LIN {X 0,Y 427.231,Z 476.03,A -85,B 0,C 180,E1 9027.625,E2 9027.625} C_VEL
LIN {X 0,Y 427.048,Z 476.03,A -85,B 0,C 180,E1 9034.562,E2 9034.562} C_VEL
LIN {X 0,Y 427.063,Z 476.03,A -85,B 0,C 180,E1 9039.656,E2 9039.656} C_VEL
LIN {X 0,Y 427.079,Z 476.03,A -85,B 0,C 180,E1 9045.158,E2 9045.158} C_VEL
LIN {X 0,Y 427.044,Z 476.03,A -85,B 0,C 180,E1 9051.263,E2 9051.263} C_VEL
LIN {X 0,Y 427.131,Z 476.03,A -85,B 0,C 180,E1 9058.294,E2 9058.294} C_VEL
LIN {X 0,Y 427.346,Z 476.125,A -85,B 0,C 180,E1 9064.803,E2 9064.803} C_VEL
LIN {X 0,Y 433.891,Z 490.356,A -85,B 0,C 180,E1 9065.954,E2 9065.954} C_VEL
LIN {X 0,Y 447.35,Z 521.334,A -85,B 0,C 180,E1 9068.749,E2 9068.749} C_VEL
LIN {X 0,Y 452.812,Z 539.377,A -85,B 0,C 180,E1 9070.383,E2 9070.383} C_VEL
LIN {X 0,Y 448.1,Z 575.713,A -85,B 0,C 180,E1 9072.93,E2 9072.93} C_VEL
LIN {X 0,Y 442.863,Z 608.573,A -85,B 0,C 180,E1 9076.154,E2 9076.154} C_VEL
LIN {X 0,Y 438.068,Z 636.216,A -85,B 0,C 180,E1 9079.797,E2 9079.797} C_VEL
LIN {X 0,Y 434.006,Z 660.175,A -85,B 0,C 180,E1 9083.993,E2 9083.993} C_VEL
LIN {X 0,Y 431.161,Z 679.406,A -85,B 0,C 180,E1 9088.491,E2 9088.491} C_VEL
LIN {X 0,Y 429.325,Z 694.838,A -85,B 0,C 180,E1 9093.539,E2 9093.539} C_VEL
LIN {X 0,Y 428.567,Z 704.775,A -85,B 0,C 180,E1 9098.423,E2 9098.423} C_VEL
LIN {X 0,Y 428.206,Z 709.346,A -85,B 0,C 180,E1 9102.249,E2 9102.249} C_VEL
LIN {X 0,Y 427.862,Z 711.472,A -85,B 0,C 180,E1 9107.165,E2 9107.165} C_VEL
LIN {X 0,Y 428.007,Z 710.105,A -85,B 0,C 180,E1 9110.718,E2 9110.718} C_VEL
LIN {X 0,Y 428.485,Z 705.369,A -85,B 0,C 180,E1 9115.09,E2 9115.09} C_VEL
LIN {X 0,Y 429.341,Z 695.552,A -85,B 0,C 180,E1 9120.096,E2 9120.096} C_VEL
LIN {X 0,Y 431.033,Z 680.185,A -85,B 0,C 180,E1 9125.219,E2 9125.219} C_VEL
LIN {X 0,Y 434.186,Z 659.155,A -85,B 0,C 180,E1 9130.146,E2 9130.146} C_VEL
LIN {X 0,Y 438.8,Z 632.297,A -85,B 0,C 180,E1 9134.712,E2 9134.712} C_VEL
LIN {X 0,Y 443.671,Z 603.64,A -85,B 0,C 180,E1 9138.309,E2 9138.309} C_VEL
LIN {X 0,Y 448.536,Z 571.756,A -85,B 0,C 180,E1 9141.287,E2 9141.287} C_VEL
LIN {X 0,Y 452.145,Z 536.862,A -85,B 0,C 180,E1 9143.702,E2 9143.702} C_VEL
LIN {X 0,Y 439.272,Z 501.491,A -85,B 0,C 180,E1 9146.972,E2 9146.972} C_VEL
LIN {X 0,Y 427.271,Z 477.331,A -85,B 0,C 180,E1 9149.227,E2 9149.227} C_VEL
LIN {X 0,Y 427.162,Z 476.03,A -85,B 0,C 180,E1 9149.465,E2 9149.465} C_VEL
LIN {X 0,Y 427.448,Z 476.03,A -85,B 0,C 180,E1 9156.294,E2 9156.294} C_VEL
LIN {X 0,Y 437.252,Z 513.904,A -85,B 0,C 180,E1 9157.675,E2 9157.675} C_VEL
LIN {X 0,Y 436.28,Z 544.603,A -85,B 0,C 180,E1 9159.138,E2 9159.138} C_VEL
LIN {X 0,Y 434.743,Z 573.454,A -85,B 0,C 180,E1 9161.342,E2 9161.342} C_VEL
LIN {X 0,Y 433.041,Z 597.944,A -85,B 0,C 180,E1 9164.095,E2 9164.095} C_VEL
LIN {X 0,Y 431.724,Z 618.004,A -85,B 0,C 180,E1 9167.336,E2 9167.336} C_VEL
LIN {X 0,Y 430.69,Z 633.102,A -85,B 0,C 180,E1 9170.895,E2 9170.895} C_VEL
LIN {X 0,Y 430.212,Z 643.735,A -85,B 0,C 180,E1 9174.949,E2 9174.949} C_VEL
LIN {X 0,Y 430.073,Z 647.839,A -85,B 0,C 180,E1 9177.979,E2 9177.979} C_VEL
LIN {X 0,Y 430.196,Z 648.552,A -85,B 0,C 180,E1 9182.014,E2 9182.014} C_VEL
LIN {X 0,Y 430.678,Z 643.75,A -85,B 0,C 180,E1 9186.051,E2 9186.051} C_VEL
LIN {X 0,Y 431.366,Z 634.554,A -85,B 0,C 180,E1 9189.594,E2 9189.594} C_VEL
LIN {X 0,Y 432.761,Z 619.622,A -85,B 0,C 180,E1 9193.141,E2 9193.141} C_VEL
LIN {X 0,Y 434.176,Z 600.487,A -85,B 0,C 180,E1 9196.195,E2 9196.195} C_VEL
LIN {X 0,Y 435.841,Z 576.008,A -85,B 0,C 180,E1 9198.871,E2 9198.871} C_VEL
LIN {X 0,Y 437.054,Z 547.742,A -85,B 0,C 180,E1 9200.91,E2 9200.91} C_VEL
LIN {X 0,Y 437.603,Z 516.913,A -85,B 0,C 180,E1 9202.249,E2 9202.249} C_VEL
LIN {X 0,Y 435.314,Z 501.555,A -85,B 0,C 180,E1 9202.759,E2 9202.759} C_VEL
LIN {X 0,Y 427.48,Z 476.03,A -85,B 0,C 180,E1 9203.775,E2 9203.775} C_VEL
LIN {X 0,Y 427.142,Z 476.03,A -85,B 0,C 180,E1 9209.747,E2 9209.747} C_VEL
LIN {X 0,Y 427.002,Z 476.03,A -85,B 0,C 180,E1 9217.064,E2 9217.064} C_VEL
LIN {X 0,Y 427.07,Z 476.03,A -85,B 0,C 180,E1 9222.339,E2 9222.339} C_VEL
LIN {X 0,Y 427.121,Z 476.674,A -85,B 0,C 180,E1 9225.541,E2 9225.541} C_VEL
LIN {X 0,Y 433.068,Z 487.614,A -85,B 0,C 180,E1 9226.618,E2 9226.618} C_VEL
LIN {X 0,Y 448.053,Z 516.786,A -85,B 0,C 180,E1 9229.257,E2 9229.257} C_VEL
LIN {X 0,Y 456.79,Z 539.614,A -85,B 0,C 180,E1 9230.965,E2 9230.965} C_VEL
LIN {X 0,Y 452.45,Z 581.575,A -85,B 0,C 180,E1 9232.645,E2 9232.645} C_VEL
LIN {X 0,Y 447.292,Z 624.098,A -85,B 0,C 180,E1 9235.225,E2 9235.225} C_VEL
LIN {X 0,Y 447.067,Z 625.988,A -85,B 0,C 180,E1 9235.366,E2 9235.366} C_VEL
LIN {X 0,Y 441.612,Z 641.029,A -85,B 0,C 180,E1 9236.319,E2 9236.319} C_VEL
LIN {X 0,Y 435.968,Z 655.399,A -85,B 0,C 180,E1 9237.373,E2 9237.373} C_VEL
LIN {X 0,Y 431.169,Z 688.074,A -85,B 0,C 180,E1 9240.997,E2 9240.997} C_VEL
LIN {X 0,Y 426.787,Z 717.547,A -85,B 0,C 180,E1 9245.363,E2 9245.363} C_VEL
LIN {X 0,Y 423.676,Z 741.475,A -85,B 0,C 180,E1 9250.153,E2 9250.153} C_VEL
LIN {X 0,Y 421.841,Z 758.815,A -85,B 0,C 180,E1 9254.916,E2 9254.916} C_VEL
LIN {X 0,Y 420.846,Z 771.829,A -85,B 0,C 180,E1 9260.16,E2 9260.16} C_VEL
LIN {X 0,Y 420.41,Z 778.626,A -85,B 0,C 180,E1 9264.834,E2 9264.834} C_VEL
LIN {X 0,Y 420.496,Z 781.231,A -85,B 0,C 180,E1 9270,E2 9270} C_VEL
LIN {X 0,Y 420.427,Z 778.636,A -85,B 0,C 180,E1 9275.165,E2 9275.165} C_VEL
LIN {X 0,Y 420.913,Z 770.827,A -85,B 0,C 180,E1 9280.361,E2 9280.361} C_VEL
LIN {X 0,Y 421.909,Z 757.336,A -85,B 0,C 180,E1 9285.614,E2 9285.614} C_VEL
LIN {X 0,Y 424.112,Z 738.412,A -85,B 0,C 180,E1 9290.643,E2 9290.643} C_VEL
LIN {X 0,Y 427.525,Z 713.526,A -85,B 0,C 180,E1 9295.452,E2 9295.452} C_VEL
LIN {X 0,Y 432.221,Z 683.275,A -85,B 0,C 180,E1 9299.788,E2 9299.788} C_VEL
LIN {X 0,Y 437.339,Z 650.056,A -85,B 0,C 180,E1 9303.34,E2 9303.34} C_VEL
LIN {X 0,Y 442.909,Z 610.784,A -85,B 0,C 180,E1 9306.426,E2 9306.426} C_VEL
LIN {X 0,Y 448.259,Z 569.03,A -85,B 0,C 180,E1 9308.695,E2 9308.695} C_VEL
LIN {X 0,Y 450.598,Z 542.743,A -85,B 0,C 180,E1 9309.738,E2 9309.738} C_VEL
LIN {X 0,Y 436.136,Z 507.763,A -85,B 0,C 180,E1 9312.473,E2 9312.473} C_VEL
LIN {X 0,Y 419.266,Z 477.454,A -85,B 0,C 180,E1 9315.25,E2 9315.25} C_VEL
LIN {X 0,Y 419.126,Z 476.03,A -85,B 0,C 180,E1 9315.373,E2 9315.373} C_VEL
LIN {X 0,Y 419.093,Z 476.03,A -85,B 0,C 180,E1 9322.638,E2 9322.638} C_VEL
LIN {X 0,Y 419.23,Z 476.03,A -85,B 0,C 180,E1 9329.633,E2 9329.633} C_VEL
LIN {X 0,Y 419.354,Z 476.03,A -85,B 0,C 180,E1 9336.604,E2 9336.604} C_VEL
LIN {X 0,Y 419.694,Z 476.03,A -85,B 0,C 180,E1 9343.23,E2 9343.23} C_VEL
LIN {X 0,Y 419.863,Z 476.03,A -85,B 0,C 180,E1 9349.616,E2 9349.616} C_VEL
LIN {X 0,Y 420.215,Z 476.03,A -85,B 0,C 180,E1 9355.871,E2 9355.871} C_VEL
LIN {X 0,Y 420.36,Z 476.03,A -85,B 0,C 180,E1 9362.067,E2 9362.067} C_VEL
LIN {X 0,Y 419.981,Z 476.03,A -85,B 0,C 180,E1 9368.294,E2 9368.294} C_VEL
LIN {X 0,Y 419.709,Z 476.03,A -85,B 0,C 180,E1 9374.629,E2 9374.629} C_VEL
LIN {X 0,Y 419.514,Z 476.03,A -85,B 0,C 180,E1 9381.159,E2 9381.159} C_VEL
LIN {X 0,Y 419.286,Z 476.03,A -85,B 0,C 180,E1 9388,E2 9388} C_VEL
LIN {X 0,Y 419.129,Z 476.03,A -85,B 0,C 180,E1 9395.311,E2 9395.311} C_VEL
LIN {X 0,Y 419.078,Z 476.03,A -85,B 0,C 180,E1 9400.649,E2 9400.649} C_VEL
LIN {X 0,Y 419.079,Z 476.03,A -85,B 0,C 180,E1 9406.65,E2 9406.65} C_VEL
LIN {X 0,Y 419.097,Z 476.03,A -85,B 0,C 180,E1 9412.638,E2 9412.638} C_VEL
LIN {X 0,Y 419.236,Z 476.03,A -85,B 0,C 180,E1 9420.086,E2 9420.086} C_VEL
LIN {X 0,Y 419.353,Z 476.296,A -85,B 0,C 180,E1 9423.929,E2 9423.929} C_VEL
LIN {X 0,Y 436.038,Z 512.102,A -85,B 0,C 180,E1 9427.125,E2 9427.125} C_VEL
LIN {X 0,Y 446.152,Z 540.478,A -85,B 0,C 180,E1 9429.827,E2 9429.827} C_VEL
LIN {X 0,Y 441.38,Z 576.647,A -85,B 0,C 180,E1 9432.404,E2 9432.404} C_VEL
LIN {X 0,Y 435.886,Z 609.52,A -85,B 0,C 180,E1 9435.671,E2 9435.671} C_VEL
LIN {X 0,Y 430.873,Z 637.095,A -85,B 0,C 180,E1 9439.369,E2 9439.369} C_VEL
LIN {X 0,Y 426.576,Z 661.024,A -85,B 0,C 180,E1 9443.632,E2 9443.632} C_VEL
LIN {X 0,Y 423.376,Z 681.097,A -85,B 0,C 180,E1 9448.463,E2 9448.463} C_VEL
LIN {X 0,Y 421.482,Z 696.246,A -85,B 0,C 180,E1 9453.605,E2 9453.605} C_VEL
LIN {X 0,Y 420.751,Z 705.431,A -85,B 0,C 180,E1 9458.277,E2 9458.277} C_VEL
LIN {X 0,Y 420.149,Z 710.82,A -85,B 0,C 180,E1 9463.345,E2 9463.345} C_VEL
LIN {X 0,Y 420.01,Z 711.669,A -85,B 0,C 180,E1 9468.932,E2 9468.932} C_VEL
LIN {X 0,Y 420.538,Z 707.058,A -85,B 0,C 180,E1 9474.46,E2 9474.46} C_VEL
LIN {X 0,Y 421.324,Z 698.418,A -85,B 0,C 180,E1 9479.398,E2 9479.398} C_VEL
LIN {X 0,Y 422.97,Z 684.165,A -85,B 0,C 180,E1 9484.58,E2 9484.58} C_VEL
LIN {X 0,Y 426.201,Z 663.636,A -85,B 0,C 180,E1 9489.752,E2 9489.752} C_VEL
LIN {X 0,Y 430.531,Z 639.285,A -85,B 0,C 180,E1 9494.212,E2 9494.212} C_VEL
LIN {X 0,Y 435.586,Z 611.344,A -85,B 0,C 180,E1 9498.027,E2 9498.027} C_VEL
LIN {X 0,Y 440.774,Z 579.985,A -85,B 0,C 180,E1 9501.212,E2 9501.212} C_VEL
LIN {X 0,Y 445.675,Z 544.214,A -85,B 0,C 180,E1 9503.835,E2 9503.835} C_VEL
LIN {X 0,Y 445.029,Z 537.901,A -85,B 0,C 180,E1 9504.333,E2 9504.333} C_VEL
LIN {X 0,Y 432.509,Z 503.331,A -85,B 0,C 180,E1 9507.658,E2 9507.658} C_VEL
LIN {X 0,Y 419.372,Z 476.912,A -85,B 0,C 180,E1 9510.248,E2 9510.248} C_VEL
LIN {X 0,Y 419.266,Z 476.03,A -85,B 0,C 180,E1 9510.489,E2 9510.489} C_VEL
LIN {X 0,Y 419.49,Z 476.03,A -85,B 0,C 180,E1 9515.93,E2 9515.93} C_VEL
LIN {X 0,Y 429.764,Z 514.336,A -85,B 0,C 180,E1 9517.345,E2 9517.345} C_VEL
LIN {X 0,Y 428.725,Z 546.754,A -85,B 0,C 180,E1 9518.922,E2 9518.922} C_VEL
LIN {X 0,Y 427.112,Z 575.273,A -85,B 0,C 180,E1 9521.16,E2 9521.16} C_VEL
LIN {X 0,Y 425.376,Z 599.612,A -85,B 0,C 180,E1 9523.959,E2 9523.959} C_VEL
LIN {X 0,Y 423.952,Z 620.118,A -85,B 0,C 180,E1 9527.362,E2 9527.362} C_VEL
LIN {X 0,Y 422.806,Z 635.929,A -85,B 0,C 180,E1 9531.28,E2 9531.28} C_VEL
LIN {X 0,Y 422.433,Z 644.927,A -85,B 0,C 180,E1 9534.856,E2 9534.856} C_VEL
LIN {X 0,Y 422.303,Z 649.133,A -85,B 0,C 180,E1 9537.942,E2 9537.942} C_VEL
LIN {X 0,Y 422.438,Z 649.948,A -85,B 0,C 180,E1 9542.051,E2 9542.051} C_VEL
LIN {X 0,Y 422.961,Z 645.197,A -85,B 0,C 180,E1 9546.161,E2 9546.161} C_VEL
LIN {X 0,Y 423.732,Z 636.039,A -85,B 0,C 180,E1 9549.768,E2 9549.768} C_VEL
LIN {X 0,Y 425.206,Z 621.071,A -85,B 0,C 180,E1 9553.379,E2 9553.379} C_VEL
LIN {X 0,Y 426.734,Z 601.915,A -85,B 0,C 180,E1 9556.486,E2 9556.486} C_VEL
LIN {X 0,Y 428.48,Z 577.271,A -85,B 0,C 180,E1 9559.208,E2 9559.208} C_VEL
LIN {X 0,Y 429.725,Z 549.886,A -85,B 0,C 180,E1 9561.224,E2 9561.224} C_VEL
LIN {X 0,Y 430.332,Z 518.139,A -85,B 0,C 180,E1 9562.626,E2 9562.626} C_VEL
LIN {X 0,Y 427.729,Z 501.755,A -85,B 0,C 180,E1 9563.195,E2 9563.195} C_VEL
LIN {X 0,Y 419.507,Z 476.03,A -85,B 0,C 180,E1 9564.342,E2 9564.342} C_VEL
LIN {X 0,Y 419.194,Z 476.03,A -85,B 0,C 180,E1 9570.37,E2 9570.37} C_VEL
LIN {X 0,Y 419.097,Z 476.03,A -85,B 0,C 180,E1 9577.361,E2 9577.361} C_VEL
LIN {X 0,Y 419.136,Z 476.03,A -85,B 0,C 180,E1 9584.353,E2 9584.353} C_VEL
LIN {X 0,Y 421.636,Z 481.766,A -85,B 0,C 180,E1 9584.893,E2 9584.893} C_VEL
LIN {X 0,Y 439.278,Z 513.737,A -85,B 0,C 180,E1 9588.19,E2 9588.19} C_VEL
LIN {X 0,Y 450.21,Z 542.434,A -85,B 0,C 180,E1 9590.458,E2 9590.458} C_VEL
LIN {X 0,Y 445.242,Z 586.094,A -85,B 0,C 180,E1 9592.329,E2 9592.329} C_VEL
LIN {X 0,Y 439.941,Z 626.973,A -85,B 0,C 180,E1 9594.943,E2 9594.943} C_VEL
LIN {X 0,Y 435.968,Z 655.399,A -85,B 0,C 180,E1 9597.373,E2 9597.373} C_VEL
LIN {X 0,Y 430.399,Z 669.303,A -85,B 0,C 180,E1 9598.572,E2 9598.572} C_VEL
LIN {X 0,Y 424.576,Z 682.557,A -85,B 0,C 180,E1 9599.9,E2 9599.9} C_VEL
LIN {X 0,Y 419.951,Z 711.698,A -85,B 0,C 180,E1 9604.077,E2 9604.077} C_VEL
LIN {X 0,Y 416.492,Z 735.835,A -85,B 0,C 180,E1 9608.682,E2 9608.682} C_VEL
LIN {X 0,Y 414.308,Z 754.62,A -85,B 0,C 180,E1 9613.547,E2 9613.547} C_VEL
LIN {X 0,Y 413.112,Z 768.969,A -85,B 0,C 180,E1 9618.906,E2 9618.906} C_VEL
LIN {X 0,Y 412.642,Z 776.819,A -85,B 0,C 180,E1 9623.68,E2 9623.68} C_VEL
LIN {X 0,Y 412.567,Z 780.149,A -85,B 0,C 180,E1 9627.896,E2 9627.896} C_VEL
LIN {X 0,Y 412.663,Z 780.169,A -85,B 0,C 180,E1 9632.102,E2 9632.102} C_VEL
LIN {X 0,Y 412.756,Z 775.793,A -85,B 0,C 180,E1 9637.173,E2 9637.173} C_VEL
LIN {X 0,Y 413.29,Z 766.728,A -85,B 0,C 180,E1 9642.16,E2 9642.16} C_VEL
LIN {X 0,Y 414.595,Z 751.858,A -85,B 0,C 180,E1 9647.368,E2 9647.368} C_VEL
LIN {X 0,Y 417.273,Z 731.307,A -85,B 0,C 180,E1 9652.426,E2 9652.426} C_VEL
LIN {X 0,Y 421.421,Z 704.435,A -85,B 0,C 180,E1 9657.264,E2 9657.264} C_VEL
LIN {X 0,Y 426.674,Z 672.562,A -85,B 0,C 180,E1 9661.503,E2 9661.503} C_VEL
LIN {X 0,Y 432.364,Z 637.205,A -85,B 0,C 180,E1 9664.967,E2 9664.967} C_VEL
LIN {X 0,Y 437.888,Z 599.138,A -85,B 0,C 180,E1 9667.696,E2 9667.696} C_VEL
LIN {X 0,Y 443.1,Z 558.883,A -85,B 0,C 180,E1 9669.697,E2 9669.697} C_VEL
LIN {X 0,Y 443.897,Z 545.511,A -85,B 0,C 180,E1 9670.263,E2 9670.263} C_VEL
LIN {X 0,Y 430.817,Z 512.727,A -85,B 0,C 180,E1 9672.888,E2 9672.888} C_VEL
LIN {X 0,Y 411.201,Z 477.084,A -85,B 0,C 180,E1 9676.286,E2 9676.286} C_VEL
LIN {X 0,Y 411.115,Z 476.03,A -85,B 0,C 180,E1 9676.579,E2 9676.579} C_VEL
LIN {X 0,Y 411.179,Z 476.03,A -85,B 0,C 180,E1 9684.107,E2 9684.107} C_VEL
LIN {X 0,Y 411.328,Z 476.03,A -85,B 0,C 180,E1 9691.416,E2 9691.416} C_VEL
LIN {X 0,Y 411.494,Z 476.03,A -85,B 0,C 180,E1 9698.416,E2 9698.416} C_VEL
LIN {X 0,Y 411.78,Z 476.03,A -85,B 0,C 180,E1 9705.089,E2 9705.089} C_VEL
LIN {X 0,Y 412.052,Z 476.03,A -85,B 0,C 180,E1 9711.552,E2 9711.552} C_VEL
LIN {X 0,Y 412.349,Z 476.03,A -85,B 0,C 180,E1 9717.899,E2 9717.899} C_VEL
LIN {X 0,Y 412.192,Z 476.03,A -85,B 0,C 180,E1 9724.216,E2 9724.216} C_VEL
LIN {X 0,Y 411.899,Z 476.03,A -85,B 0,C 180,E1 9730.594,E2 9730.594} C_VEL
LIN {X 0,Y 411.721,Z 476.03,A -85,B 0,C 180,E1 9737.112,E2 9737.112} C_VEL
LIN {X 0,Y 411.487,Z 476.03,A -85,B 0,C 180,E1 9743.878,E2 9743.878} C_VEL
LIN {X 0,Y 411.356,Z 476.03,A -85,B 0,C 180,E1 9748.589,E2 9748.589} C_VEL
LIN {X 0,Y 411.182,Z 476.03,A -85,B 0,C 180,E1 9756.099,E2 9756.099} C_VEL
LIN {X 0,Y 411.091,Z 476.03,A -85,B 0,C 180,E1 9762.555,E2 9762.555} C_VEL
LIN {X 0,Y 411.102,Z 476.03,A -85,B 0,C 180,E1 9768.475,E2 9768.475} C_VEL
LIN {X 0,Y 411.141,Z 476.03,A -85,B 0,C 180,E1 9774.115,E2 9774.115} C_VEL
LIN {X 0,Y 411.332,Z 476.03,A -85,B 0,C 180,E1 9781.411,E2 9781.411} C_VEL
LIN {X 0,Y 411.384,Z 476.03,A -85,B 0,C 180,E1 9783.001,E2 9783.001} C_VEL
LIN {X 0,Y 415.875,Z 486.011,A -85,B 0,C 180,E1 9783.845,E2 9783.845} C_VEL
LIN {X 0,Y 430.593,Z 517.419,A -85,B 0,C 180,E1 9786.841,E2 9786.841} C_VEL
LIN {X 0,Y 439.499,Z 543.425,A -85,B 0,C 180,E1 9789.39,E2 9789.39} C_VEL
LIN {X 0,Y 434.466,Z 578.892,A -85,B 0,C 180,E1 9791.984,E2 9791.984} C_VEL
LIN {X 0,Y 428.954,Z 610.397,A -85,B 0,C 180,E1 9795.173,E2 9795.173} C_VEL
LIN {X 0,Y 423.704,Z 637.986,A -85,B 0,C 180,E1 9798.926,E2 9798.926} C_VEL
LIN {X 0,Y 419.119,Z 661.865,A -85,B 0,C 180,E1 9803.258,E2 9803.258} C_VEL
LIN {X 0,Y 415.902,Z 680.983,A -85,B 0,C 180,E1 9807.914,E2 9807.914} C_VEL
LIN {X 0,Y 413.8,Z 696.37,A -85,B 0,C 180,E1 9813.147,E2 9813.147} C_VEL
LIN {X 0,Y 412.869,Z 706.505,A -85,B 0,C 180,E1 9818.436,E2 9818.436} C_VEL
LIN {X 0,Y 412.38,Z 711.13,A -85,B 0,C 180,E1 9822.727,E2 9822.727} C_VEL
LIN {X 0,Y 412.099,Z 712.634,A -85,B 0,C 180,E1 9827.202,E2 9827.202} C_VEL
LIN {X 0,Y 412.327,Z 710.876,A -85,B 0,C 180,E1 9831.544,E2 9831.544} C_VEL
LIN {X 0,Y 412.906,Z 705.62,A -85,B 0,C 180,E1 9836.107,E2 9836.107} C_VEL
LIN {X 0,Y 414.174,Z 693.785,A -85,B 0,C 180,E1 9841.831,E2 9841.831} C_VEL
LIN {X 0,Y 416.551,Z 677.122,A -85,B 0,C 180,E1 9847.088,E2 9847.088} C_VEL
LIN {X 0,Y 420.489,Z 654.97,A -85,B 0,C 180,E1 9852.059,E2 9852.059} C_VEL
LIN {X 0,Y 425.795,Z 627.465,A -85,B 0,C 180,E1 9856.569,E2 9856.569} C_VEL
LIN {X 0,Y 431.511,Z 596.399,A -85,B 0,C 180,E1 9860.296,E2 9860.296} C_VEL
LIN {X 0,Y 436.907,Z 562.912,A -85,B 0,C 180,E1 9863.216,E2 9863.216} C_VEL
LIN {X 0,Y 438.983,Z 542.389,A -85,B 0,C 180,E1 9864.651,E2 9864.651} C_VEL
LIN {X 0,Y 427.209,Z 508.437,A -85,B 0,C 180,E1 9868.045,E2 9868.045} C_VEL
LIN {X 0,Y 413.155,Z 481.024,A -85,B 0,C 180,E1 9870.964,E2 9870.964} C_VEL
LIN {X 0,Y 411.367,Z 476.03,A -85,B 0,C 180,E1 9871.412,E2 9871.412} C_VEL
LIN {X 0,Y 411.566,Z 476.03,A -85,B 0,C 180,E1 9875.515,E2 9875.515} C_VEL
LIN {X 0,Y 422.237,Z 516.448,A -85,B 0,C 180,E1 9877.069,E2 9877.069} C_VEL
LIN {X 0,Y 421.211,Z 547.714,A -85,B 0,C 180,E1 9878.629,E2 9878.629} C_VEL
LIN {X 0,Y 419.509,Z 576.636,A -85,B 0,C 180,E1 9880.934,E2 9880.934} C_VEL
LIN {X 0,Y 417.634,Z 602.098,A -85,B 0,C 180,E1 9883.945,E2 9883.945} C_VEL
LIN {X 0,Y 416.183,Z 622.169,A -85,B 0,C 180,E1 9887.389,E2 9887.389} C_VEL
LIN {X 0,Y 415.05,Z 637.085,A -85,B 0,C 180,E1 9891.158,E2 9891.158} C_VEL
LIN {X 0,Y 414.648,Z 646.108,A -85,B 0,C 180,E1 9894.759,E2 9894.759} C_VEL
LIN {X 0,Y 414.544,Z 650.422,A -85,B 0,C 180,E1 9897.904,E2 9897.904} C_VEL
LIN {X 0,Y 414.678,Z 651.347,A -85,B 0,C 180,E1 9902.089,E2 9902.089} C_VEL
LIN {X 0,Y 415.271,Z 646.676,A -85,B 0,C 180,E1 9906.276,E2 9906.276} C_VEL
LIN {X 0,Y 416.085,Z 637.535,A -85,B 0,C 180,E1 9909.95,E2 9909.95} C_VEL
LIN {X 0,Y 417.664,Z 622.596,A -85,B 0,C 180,E1 9913.625,E2 9913.625} C_VEL
LIN {X 0,Y 419.307,Z 603.371,A -85,B 0,C 180,E1 9916.786,E2 9916.786} C_VEL
LIN {X 0,Y 421.157,Z 578.664,A -85,B 0,C 180,E1 9919.555,E2 9919.555} C_VEL
LIN {X 0,Y 422.545,Z 549.776,A -85,B 0,C 180,E1 9921.681,E2 9921.681} C_VEL
LIN {X 0,Y 423.126,Z 519.185,A -85,B 0,C 180,E1 9923.033,E2 9923.033} C_VEL
LIN {X 0,Y 420.255,Z 502.359,A -85,B 0,C 180,E1 9923.645,E2 9923.645} C_VEL
LIN {X 0,Y 411.561,Z 476.03,A -85,B 0,C 180,E1 9924.958,E2 9924.958} C_VEL
LIN {X 0,Y 411.158,Z 476.03,A -85,B 0,C 180,E1 9932.113,E2 9932.113} C_VEL
LIN {X 0,Y 411.091,Z 476.03,A -85,B 0,C 180,E1 9938.758,E2 9938.758} C_VEL
LIN {X 0,Y 411.143,Z 476.03,A -85,B 0,C 180,E1 9943.126,E2 9943.126} C_VEL
LIN {X 0,Y 413.592,Z 481.72,A -85,B 0,C 180,E1 9943.703,E2 9943.703} C_VEL
LIN {X 0,Y 431.305,Z 512.933,A -85,B 0,C 180,E1 9947.228,E2 9947.228} C_VEL
LIN {X 0,Y 438.697,Z 531.693,A -85,B 0,C 180,E1 9948.831,E2 9948.831} C_VEL
LIN {X 0,Y 443.478,Z 546.408,A -85,B 0,C 180,E1 9949.979,E2 9949.979} C_VEL
LIN {X 0,Y 438.302,Z 589.006,A -85,B 0,C 180,E1 9951.917,E2 9951.917} C_VEL
LIN {X 0,Y 432.451,Z 630.665,A -85,B 0,C 180,E1 9954.71,E2 9954.71} C_VEL
LIN {X 0,Y 426.772,Z 668.295,A -85,B 0,C 180,E1 9958.234,E2 9958.234} C_VEL
LIN {X 0,Y 424.576,Z 682.557,A -85,B 0,C 180,E1 9959.9,E2 9959.9} C_VEL
LIN {X 0,Y 418.716,Z 695.182,A -85,B 0,C 180,E1 9961.365,E2 9961.365} C_VEL
LIN {X 0,Y 413.148,Z 707.004,A -85,B 0,C 180,E1 9962.969,E2 9962.969} C_VEL
LIN {X 0,Y 409.316,Z 731.965,A -85,B 0,C 180,E1 9967.617,E2 9967.617} C_VEL
LIN {X 0,Y 406.712,Z 752.02,A -85,B 0,C 180,E1 9972.673,E2 9972.673} C_VEL
LIN {X 0,Y 405.272,Z 767.081,A -85,B 0,C 180,E1 9978.142,E2 9978.142} C_VEL
LIN {X 0,Y 404.776,Z 776.139,A -85,B 0,C 180,E1 9983.556,E2 9983.556} C_VEL
LIN {X 0,Y 404.684,Z 779.491,A -85,B 0,C 180,E1 9987.855,E2 9987.855} C_VEL
LIN {X 0,Y 404.778,Z 779.523,A -85,B 0,C 180,E1 9992.143,E2 9992.143} C_VEL
LIN {X 0,Y 404.902,Z 774.393,A -85,B 0,C 180,E1 9997.864,E2 9997.864} C_VEL
LIN {X 0,Y 405.515,Z 764.81,A -85,B 0,C 180,E1 10002.945,E2 10002.945} C_VEL
LIN {X 0,Y 407.126,Z 748.885,A -85,B 0,C 180,E1 10008.369,E2 10008.369} C_VEL
LIN {X 0,Y 410.144,Z 727.387,A -85,B 0,C 180,E1 10013.516,E2 10013.516} C_VEL
LIN {X 0,Y 414.38,Z 701.736,A -85,B 0,C 180,E1 10018.063,E2 10018.063} C_VEL
LIN {X 0,Y 419.901,Z 670.053,A -85,B 0,C 180,E1 10022.256,E2 10022.256} C_VEL
LIN {X 0,Y 425.92,Z 633.952,A -85,B 0,C 180,E1 10025.756,E2 10025.756} C_VEL
LIN {X 0,Y 431.625,Z 596.138,A -85,B 0,C 180,E1 10028.443,E2 10028.443} C_VEL
LIN {X 0,Y 437.186,Z 554.886,A -85,B 0,C 180,E1 10030.458,E2 10030.458} C_VEL
LIN {X 0,Y 437.077,Z 548.035,A -85,B 0,C 180,E1 10030.798,E2 10030.798} C_VEL
LIN {X 0,Y 425.443,Z 517.565,A -85,B 0,C 180,E1 10033.315,E2 10033.315} C_VEL
LIN {X 0,Y 403.219,Z 477.051,A -85,B 0,C 180,E1 10037.352,E2 10037.352} C_VEL
LIN {X 0,Y 403.143,Z 476.03,A -85,B 0,C 180,E1 10037.473,E2 10037.473} C_VEL
LIN {X 0,Y 403.137,Z 476.03,A -85,B 0,C 180,E1 10043.071,E2 10043.071} C_VEL
LIN {X 0,Y 403.289,Z 476.03,A -85,B 0,C 180,E1 10049.713,E2 10049.713} C_VEL
LIN {X 0,Y 403.433,Z 476.03,A -85,B 0,C 180,E1 10055.622,E2 10055.622} C_VEL
LIN {X 0,Y 403.787,Z 476.03,A -85,B 0,C 180,E1 10062.548,E2 10062.548} C_VEL
LIN {X 0,Y 403.994,Z 476.03,A -85,B 0,C 180,E1 10069.203,E2 10069.203} C_VEL
LIN {X 0,Y 404.375,Z 476.03,A -85,B 0,C 180,E1 10075.709,E2 10075.709} C_VEL
LIN {X 0,Y 404.551,Z 476.03,A -85,B 0,C 180,E1 10082.148,E2 10082.148} C_VEL
LIN {X 0,Y 404.128,Z 476.03,A -85,B 0,C 180,E1 10088.622,E2 10088.622} C_VEL
LIN {X 0,Y 403.827,Z 476.03,A -85,B 0,C 180,E1 10095.218,E2 10095.218} C_VEL
LIN {X 0,Y 403.62,Z 476.03,A -85,B 0,C 180,E1 10102.034,E2 10102.034} C_VEL
LIN {X 0,Y 403.352,Z 476.03,A -85,B 0,C 180,E1 10109.211,E2 10109.211} C_VEL
LIN {X 0,Y 403.238,Z 476.03,A -85,B 0,C 180,E1 10114.303,E2 10114.303} C_VEL
LIN {X 0,Y 403.164,Z 476.03,A -85,B 0,C 180,E1 10121.313,E2 10121.313} C_VEL
LIN {X 0,Y 403.207,Z 476.03,A -85,B 0,C 180,E1 10127.474,E2 10127.474} C_VEL
LIN {X 0,Y 403.142,Z 476.03,A -85,B 0,C 180,E1 10133.064,E2 10133.064} C_VEL
LIN {X 0,Y 403.268,Z 476.03,A -85,B 0,C 180,E1 10139.718,E2 10139.718} C_VEL
LIN {X 0,Y 403.479,Z 476.03,A -85,B 0,C 180,E1 10142.063,E2 10142.063} C_VEL
LIN {X 0,Y 408.04,Z 486.236,A -85,B 0,C 180,E1 10142.944,E2 10142.944} C_VEL
LIN {X 0,Y 422.577,Z 516.877,A -85,B 0,C 180,E1 10145.959,E2 10145.959} C_VEL
LIN {X 0,Y 432.598,Z 545.242,A -85,B 0,C 180,E1 10148.837,E2 10148.837} C_VEL
LIN {X 0,Y 427.592,Z 581.067,A -85,B 0,C 180,E1 10151.55,E2 10151.55} C_VEL
LIN {X 0,Y 421.673,Z 613.313,A -85,B 0,C 180,E1 10154.911,E2 10154.911} C_VEL
LIN {X 0,Y 415.886,Z 642.006,A -85,B 0,C 180,E1 10158.981,E2 10158.981} C_VEL
LIN {X 0,Y 411.053,Z 666.335,A -85,B 0,C 180,E1 10163.656,E2 10163.656} C_VEL
LIN {X 0,Y 407.567,Z 686.188,A -85,B 0,C 180,E1 10168.936,E2 10168.936} C_VEL
LIN {X 0,Y 405.714,Z 700.138,A -85,B 0,C 180,E1 10174.281,E2 10174.281} C_VEL
LIN {X 0,Y 404.867,Z 709.002,A -85,B 0,C 180,E1 10179.689,E2 10179.689} C_VEL
LIN {X 0,Y 404.275,Z 713.033,A -85,B 0,C 180,E1 10185.199,E2 10185.199} C_VEL
LIN {X 0,Y 404.33,Z 712.238,A -85,B 0,C 180,E1 10190.581,E2 10190.581} C_VEL
LIN {X 0,Y 405.088,Z 706.371,A -85,B 0,C 180,E1 10196.227,E2 10196.227} C_VEL
LIN {X 0,Y 406.418,Z 694.871,A -85,B 0,C 180,E1 10201.943,E2 10201.943} C_VEL
LIN {X 0,Y 408.926,Z 678.237,A -85,B 0,C 180,E1 10207.337,E2 10207.337} C_VEL
LIN {X 0,Y 412.881,Z 657.372,A -85,B 0,C 180,E1 10212.172,E2 10212.172} C_VEL
LIN {X 0,Y 417.988,Z 632.122,A -85,B 0,C 180,E1 10216.508,E2 10216.508} C_VEL
LIN {X 0,Y 423.969,Z 601.754,A -85,B 0,C 180,E1 10220.375,E2 10220.375} C_VEL
LIN {X 0,Y 429.741,Z 568.805,A -85,B 0,C 180,E1 10223.437,E2 10223.437} C_VEL
LIN {X 0,Y 432.739,Z 546.087,A -85,B 0,C 180,E1 10225.055,E2 10225.055} C_VEL
LIN {X 0,Y 421.075,Z 511.505,A -85,B 0,C 180,E1 10228.648,E2 10228.648} C_VEL
LIN {X 0,Y 406.053,Z 481.876,A -85,B 0,C 180,E1 10231.955,E2 10231.955} C_VEL
LIN {X 0,Y 403.442,Z 476.03,A -85,B 0,C 180,E1 10232.602,E2 10232.602} C_VEL
LIN {X 0,Y 403.625,Z 476.03,A -85,B 0,C 180,E1 10235.109,E2 10235.109} C_VEL
LIN {X 0,Y 414.766,Z 517.074,A -85,B 0,C 180,E1 10236.728,E2 10236.728} C_VEL
LIN {X 0,Y 413.673,Z 549.158,A -85,B 0,C 180,E1 10238.355,E2 10238.355} C_VEL
LIN {X 0,Y 411.931,Z 577.802,A -85,B 0,C 180,E1 10240.68,E2 10240.68} C_VEL
LIN {X 0,Y 410.039,Z 602.613,A -85,B 0,C 180,E1 10243.641,E2 10243.641} C_VEL
LIN {X 0,Y 408.499,Z 622.961,A -85,B 0,C 180,E1 10247.148,E2 10247.148} C_VEL
LIN {X 0,Y 407.284,Z 638.382,A -85,B 0,C 180,E1 10251.08,E2 10251.08} C_VEL
LIN {X 0,Y 406.869,Z 647.278,A -85,B 0,C 180,E1 10254.659,E2 10254.659} C_VEL
LIN {X 0,Y 406.763,Z 651.709,A -85,B 0,C 180,E1 10257.864,E2 10257.864} C_VEL
LIN {X 0,Y 406.919,Z 652.758,A -85,B 0,C 180,E1 10262.129,E2 10262.129} C_VEL
LIN {X 0,Y 407.57,Z 648.158,A -85,B 0,C 180,E1 10266.395,E2 10266.395} C_VEL
LIN {X 0,Y 408.479,Z 639.077,A -85,B 0,C 180,E1 10270.137,E2 10270.137} C_VEL
LIN {X 0,Y 410.137,Z 624.133,A -85,B 0,C 180,E1 10273.88,E2 10273.88} C_VEL
LIN {X 0,Y 411.928,Z 604.752,A -85,B 0,C 180,E1 10277.121,E2 10277.121} C_VEL
LIN {X 0,Y 413.85,Z 580.689,A -85,B 0,C 180,E1 10279.863,E2 10279.863} C_VEL
LIN {X 0,Y 415.25,Z 552.643,A -85,B 0,C 180,E1 10281.992,E2 10281.992} C_VEL
LIN {X 0,Y 415.964,Z 520.456,A -85,B 0,C 180,E1 10283.458,E2 10283.458} C_VEL
LIN {X 0,Y 412.931,Z 503.212,A -85,B 0,C 180,E1 10284.111,E2 10284.111} C_VEL
LIN {X 0,Y 403.588,Z 476.03,A -85,B 0,C 180,E1 10285.56,E2 10285.56} C_VEL
LIN {X 0,Y 403.264,Z 476.03,A -85,B 0,C 180,E1 10291.706,E2 10291.706} C_VEL
LIN {X 0,Y 403.117,Z 476.03,A -85,B 0,C 180,E1 10297.929,E2 10297.929} C_VEL
LIN {X 0,Y 403.203,Z 476.03,A -85,B 0,C 180,E1 10301.794,E2 10301.794} C_VEL
LIN {X 0,Y 405.715,Z 481.812,A -85,B 0,C 180,E1 10302.459,E2 10302.459} C_VEL
LIN {X 0,Y 422.633,Z 510.989,A -85,B 0,C 180,E1 10306.06,E2 10306.06} C_VEL
LIN {X 0,Y 431.817,Z 532.148,A -85,B 0,C 180,E1 10308.084,E2 10308.084} C_VEL
LIN {X 0,Y 436.945,Z 548.625,A -85,B 0,C 180,E1 10309.431,E2 10309.431} C_VEL
LIN {X 0,Y 431.399,Z 591.47,A -85,B 0,C 180,E1 10311.474,E2 10311.474} C_VEL
LIN {X 0,Y 425.256,Z 632.56,A -85,B 0,C 180,E1 10314.336,E2 10314.336} C_VEL
LIN {X 0,Y 419.481,Z 668.892,A -85,B 0,C 180,E1 10317.835,E2 10317.835} C_VEL
LIN {X 0,Y 414.301,Z 700.31,A -85,B 0,C 180,E1 10321.931,E2 10321.931} C_VEL
LIN {X 0,Y 413.148,Z 707.004,A -85,B 0,C 180,E1 10322.969,E2 10322.969} C_VEL
LIN {X 0,Y 407.604,Z 718.074,A -85,B 0,C 180,E1 10324.705,E2 10324.705} C_VEL
LIN {X 0,Y 402.105,Z 728.309,A -85,B 0,C 180,E1 10326.574,E2 10326.574} C_VEL
LIN {X 0,Y 399.203,Z 749.578,A -85,B 0,C 180,E1 10331.84,E2 10331.84} C_VEL
LIN {X 0,Y 397.506,Z 765.098,A -85,B 0,C 180,E1 10337.348,E2 10337.348} C_VEL
LIN {X 0,Y 396.935,Z 774.436,A -85,B 0,C 180,E1 10342.587,E2 10342.587} C_VEL
LIN {X 0,Y 396.802,Z 778.833,A -85,B 0,C 180,E1 10347.813,E2 10347.813} C_VEL
LIN {X 0,Y 396.893,Z 778.877,A -85,B 0,C 180,E1 10352.186,E2 10352.186} C_VEL
LIN {X 0,Y 396.982,Z 774.498,A -85,B 0,C 180,E1 10357.465,E2 10357.465} C_VEL
LIN {X 0,Y 397.596,Z 765.387,A -85,B 0,C 180,E1 10362.648,E2 10362.648} C_VEL
LIN {X 0,Y 399.159,Z 750.205,A -85,B 0,C 180,E1 10368.129,E2 10368.129} C_VEL
LIN {X 0,Y 402.034,Z 730.131,A -85,B 0,C 180,E1 10373.236,E2 10373.236} C_VEL
LIN {X 0,Y 406.495,Z 704.332,A -85,B 0,C 180,E1 10378.051,E2 10378.051} C_VEL
LIN {X 0,Y 411.826,Z 674.884,A -85,B 0,C 180,E1 10382.164,E2 10382.164} C_VEL
LIN {X 0,Y 417.951,Z 640.364,A -85,B 0,C 180,E1 10385.743,E2 10385.743} C_VEL
LIN {X 0,Y 423.992,Z 602.414,A -85,B 0,C 180,E1 10388.63,E2 10388.63} C_VEL
LIN {X 0,Y 429.923,Z 561.523,A -85,B 0,C 180,E1 10390.802,E2 10390.802} C_VEL
LIN {X 0,Y 430.652,Z 551.335,A -85,B 0,C 180,E1 10391.275,E2 10391.275} C_VEL
LIN {X 0,Y 420.148,Z 522.666,A -85,B 0,C 180,E1 10393.7,E2 10393.7} C_VEL
LIN {X 0,Y 397.602,Z 481.679,A -85,B 0,C 180,E1 10397.994,E2 10397.994} C_VEL
LIN {X 0,Y 395.208,Z 476.03,A -85,B 0,C 180,E1 10398.53,E2 10398.53} C_VEL
LIN {X 0,Y 395.248,Z 476.03,A -85,B 0,C 180,E1 10404.934,E2 10404.934} C_VEL
LIN {X 0,Y 395.389,Z 476.03,A -85,B 0,C 180,E1 10411.735,E2 10411.735} C_VEL
LIN {X 0,Y 395.569,Z 476.03,A -85,B 0,C 180,E1 10417.5,E2 10417.5} C_VEL
LIN {X 0,Y 395.897,Z 476.03,A -85,B 0,C 180,E1 10424.476,E2 10424.476} C_VEL
LIN {X 0,Y 396.193,Z 476.03,A -85,B 0,C 180,E1 10431.211,E2 10431.211} C_VEL
LIN {X 0,Y 396.557,Z 476.03,A -85,B 0,C 180,E1 10437.815,E2 10437.815} C_VEL
LIN {X 0,Y 396.368,Z 476.03,A -85,B 0,C 180,E1 10444.385,E2 10444.385} C_VEL
LIN {X 0,Y 396.04,Z 476.03,A -85,B 0,C 180,E1 10451.023,E2 10451.023} C_VEL
LIN {X 0,Y 395.814,Z 476.03,A -85,B 0,C 180,E1 10457.822,E2 10457.822} C_VEL
LIN {X 0,Y 395.568,Z 476.03,A -85,B 0,C 180,E1 10464.902,E2 10464.902} C_VEL
LIN {X 0,Y 395.422,Z 476.03,A -85,B 0,C 180,E1 10469.855,E2 10469.855} C_VEL
LIN {X 0,Y 395.223,Z 476.03,A -85,B 0,C 180,E1 10476.437,E2 10476.437} C_VEL
LIN {X 0,Y 395.241,Z 476.03,A -85,B 0,C 180,E1 10483.596,E2 10483.596} C_VEL
LIN {X 0,Y 395.255,Z 476.03,A -85,B 0,C 180,E1 10490.009,E2 10490.009} C_VEL
LIN {X 0,Y 395.272,Z 476.03,A -85,B 0,C 180,E1 10497.57,E2 10497.57} C_VEL
LIN {X 0,Y 395.471,Z 476.366,A -85,B 0,C 180,E1 10501.07,E2 10501.07} C_VEL
LIN {X 0,Y 403.174,Z 491.824,A -85,B 0,C 180,E1 10502.557,E2 10502.557} C_VEL
LIN {X 0,Y 417.789,Z 523.894,A -85,B 0,C 180,E1 10505.829,E2 10505.829} C_VEL
LIN {X 0,Y 425.946,Z 549.703,A -85,B 0,C 180,E1 10508.51,E2 10508.51} C_VEL
LIN {X 0,Y 420.708,Z 583.185,A -85,B 0,C 180,E1 10511.101,E2 10511.101} C_VEL
LIN {X 0,Y 414.768,Z 614.107,A -85,B 0,C 180,E1 10514.382,E2 10514.382} C_VEL
LIN {X 0,Y 408.741,Z 642.83,A -85,B 0,C 180,E1 10518.516,E2 10518.516} C_VEL
LIN {X 0,Y 403.628,Z 667.144,A -85,B 0,C 180,E1 10523.268,E2 10523.268} C_VEL
LIN {X 0,Y 400.059,Z 686.161,A -85,B 0,C 180,E1 10528.374,E2 10528.374} C_VEL
LIN {X 0,Y 397.98,Z 700.35,A -85,B 0,C 180,E1 10533.818,E2 10533.818} C_VEL
LIN {X 0,Y 397.117,Z 708.649,A -85,B 0,C 180,E1 10538.773,E2 10538.773} C_VEL
LIN {X 0,Y 396.555,Z 712.862,A -85,B 0,C 180,E1 10543.244,E2 10543.244} C_VEL
LIN {X 0,Y 396.346,Z 713.845,A -85,B 0,C 180,E1 10547.796,E2 10547.796} C_VEL
LIN {X 0,Y 396.846,Z 710.382,A -85,B 0,C 180,E1 10553.697,E2 10553.697} C_VEL
LIN {X 0,Y 397.743,Z 702.786,A -85,B 0,C 180,E1 10558.89,E2 10558.89} C_VEL
LIN {X 0,Y 399.399,Z 690.912,A -85,B 0,C 180,E1 10563.971,E2 10563.971} C_VEL
LIN {X 0,Y 402.666,Z 672.38,A -85,B 0,C 180,E1 10569.429,E2 10569.429} C_VEL
LIN {X 0,Y 407.404,Z 649.633,A -85,B 0,C 180,E1 10574.258,E2 10574.258} C_VEL
LIN {X 0,Y 413.391,Z 621.776,A -85,B 0,C 180,E1 10578.62,E2 10578.62} C_VEL
LIN {X 0,Y 419.766,Z 589.599,A -85,B 0,C 180,E1 10582.304,E2 10582.304} C_VEL
LIN {X 0,Y 425.538,Z 554.641,A -85,B 0,C 180,E1 10585.167,E2 10585.167} C_VEL
LIN {X 0,Y 425.924,Z 547.747,A -85,B 0,C 180,E1 10585.696,E2 10585.696} C_VEL
LIN {X 0,Y 414.973,Z 514.564,A -85,B 0,C 180,E1 10589.28,E2 10589.28} C_VEL
LIN {X 0,Y 401.337,Z 487.343,A -85,B 0,C 180,E1 10592.472,E2 10592.472} C_VEL
LIN {X 0,Y 395.61,Z 476.934,A -85,B 0,C 180,E1 10593.783,E2 10593.783} C_VEL
LIN {X 0,Y 395.628,Z 476.03,A -85,B 0,C 180,E1 10594.444,E2 10594.444} C_VEL
LIN {X 0,Y 395.667,Z 476.03,A -85,B 0,C 180,E1 10594.715,E2 10594.715} C_VEL
LIN {X 0,Y 407.176,Z 517.659,A -85,B 0,C 180,E1 10596.379,E2 10596.379} C_VEL
LIN {X 0,Y 406.179,Z 549.675,A -85,B 0,C 180,E1 10598.023,E2 10598.023} C_VEL
LIN {X 0,Y 404.316,Z 579.127,A -85,B 0,C 180,E1 10600.444,E2 10600.444} C_VEL
LIN {X 0,Y 402.317,Z 604.218,A -85,B 0,C 180,E1 10603.498,E2 10603.498} C_VEL
LIN {X 0,Y 400.717,Z 624.98,A -85,B 0,C 180,E1 10607.172,E2 10607.172} C_VEL
LIN {X 0,Y 399.5,Z 640.495,A -85,B 0,C 180,E1 10611.278,E2 10611.278} C_VEL
LIN {X 0,Y 399.126,Z 650.298,A -85,B 0,C 180,E1 10615.646,E2 10615.646} C_VEL
LIN {X 0,Y 399.127,Z 654.259,A -85,B 0,C 180,E1 10619.997,E2 10619.997} C_VEL
LIN {X 0,Y 399.389,Z 652.661,A -85,B 0,C 180,E1 10624.345,E2 10624.345} C_VEL
LIN {X 0,Y 400.385,Z 645.151,A -85,B 0,C 180,E1 10628.696,E2 10628.696} C_VEL
LIN {X 0,Y 401.963,Z 631.933,A -85,B 0,C 180,E1 10632.753,E2 10632.753} C_VEL
LIN {X 0,Y 403.882,Z 613.455,A -85,B 0,C 180,E1 10636.369,E2 10636.369} C_VEL
LIN {X 0,Y 405.876,Z 591.113,A -85,B 0,C 180,E1 10639.329,E2 10639.329} C_VEL
LIN {X 0,Y 407.659,Z 563.435,A -85,B 0,C 180,E1 10641.798,E2 10641.798} C_VEL
LIN {X 0,Y 408.676,Z 532.217,A -85,B 0,C 180,E1 10643.521,E2 10643.521} C_VEL
LIN {X 0,Y 407.871,Z 512.659,A -85,B 0,C 180,E1 10644.244,E2 10644.244} C_VEL
LIN {X 0,Y 398.716,Z 484.45,A -85,B 0,C 180,E1 10645.674,E2 10645.674} C_VEL
LIN {X 0,Y 395.571,Z 476.03,A -85,B 0,C 180,E1 10646.263,E2 10646.263} C_VEL
LIN {X 0,Y 395.285,Z 476.03,A -85,B 0,C 180,E1 10652.573,E2 10652.573} C_VEL
LIN {X 0,Y 395.251,Z 476.03,A -85,B 0,C 180,E1 10659.989,E2 10659.989} C_VEL
LIN {X 0,Y 395.257,Z 476.752,A -85,B 0,C 180,E1 10660.446,E2 10660.446} C_VEL
LIN {X 0,Y 398.25,Z 482.217,A -85,B 0,C 180,E1 10661.198,E2 10661.198} C_VEL
LIN {X 0,Y 416.522,Z 513.903,A -85,B 0,C 180,E1 10665.364,E2 10665.364} C_VEL
LIN {X 0,Y 425.985,Z 535.928,A -85,B 0,C 180,E1 10667.587,E2 10667.587} C_VEL
LIN {X 0,Y 430.396,Z 551.645,A -85,B 0,C 180,E1 10668.887,E2 10668.887} C_VEL
LIN {X 0,Y 424.199,Z 596.388,A -85,B 0,C 180,E1 10671.16,E2 10671.16} C_VEL
LIN {X 0,Y 417.564,Z 637.75,A -85,B 0,C 180,E1 10674.217,E2 10674.217} C_VEL
LIN {X 0,Y 411.398,Z 673.898,A -85,B 0,C 180,E1 10677.931,E2 10677.931} C_VEL
LIN {X 0,Y 406.048,Z 704.655,A -85,B 0,C 180,E1 10682.217,E2 10682.217} C_VEL
LIN {X 0,Y 402.105,Z 728.309,A -85,B 0,C 180,E1 10686.574,E2 10686.574} C_VEL
LIN {X 0,Y 396.812,Z 737.667,A -85,B 0,C 180,E1 10688.565,E2 10688.565} C_VEL
LIN {X 0,Y 391.808,Z 746.088,A -85,B 0,C 180,E1 10690.685,E2 10690.685} C_VEL
LIN {X 0,Y 389.937,Z 762.013,A -85,B 0,C 180,E1 10696.075,E2 10696.075} C_VEL
LIN {X 0,Y 389.186,Z 771.794,A -85,B 0,C 180,E1 10701.047,E2 10701.047} C_VEL
LIN {X 0,Y 388.909,Z 776.892,A -85,B 0,C 180,E1 10705.534,E2 10705.534} C_VEL
LIN {X 0,Y 388.997,Z 778.637,A -85,B 0,C 180,E1 10710,E2 10710} C_VEL
LIN {X 0,Y 388.956,Z 776.06,A -85,B 0,C 180,E1 10715.584,E2 10715.584} C_VEL
LIN {X 0,Y 389.487,Z 768.202,A -85,B 0,C 180,E1 10721.208,E2 10721.208} C_VEL
LIN {X 0,Y 390.735,Z 754.506,A -85,B 0,C 180,E1 10726.895,E2 10726.895} C_VEL
LIN {X 0,Y 393.489,Z 735.273,A -85,B 0,C 180,E1 10732.332,E2 10732.332} C_VEL
LIN {X 0,Y 397.642,Z 711.767,A -85,B 0,C 180,E1 10737.189,E2 10737.189} C_VEL
LIN {X 0,Y 403.41,Z 681.234,A -85,B 0,C 180,E1 10741.851,E2 10741.851} C_VEL
LIN {X 0,Y 409.637,Z 647.683,A -85,B 0,C 180,E1 10745.604,E2 10745.604} C_VEL
LIN {X 0,Y 416.342,Z 608.598,A -85,B 0,C 180,E1 10748.807,E2 10748.807} C_VEL
LIN {X 0,Y 422.729,Z 567.013,A -85,B 0,C 180,E1 10751.177,E2 10751.177} C_VEL
LIN {X 0,Y 424.258,Z 554.656,A -85,B 0,C 180,E1 10751.733,E2 10751.733} C_VEL
LIN {X 0,Y 414.401,Z 527.034,A -85,B 0,C 180,E1 10754.159,E2 10754.159} C_VEL
LIN {X 0,Y 392.863,Z 487.24,A -85,B 0,C 180,E1 10758.477,E2 10758.477} C_VEL
LIN {X 0,Y 387.39,Z 477.155,A -85,B 0,C 180,E1 10759.604,E2 10759.604} C_VEL
LIN {X 0,Y 387.296,Z 476.03,A -85,B 0,C 180,E1 10759.661,E2 10759.661} C_VEL
LIN {X 0,Y 387.348,Z 476.03,A -85,B 0,C 180,E1 10766.828,E2 10766.828} C_VEL
LIN {X 0,Y 387.489,Z 476.03,A -85,B 0,C 180,E1 10773.99,E2 10773.99} C_VEL
LIN {X 0,Y 387.78,Z 476.03,A -85,B 0,C 180,E1 10779.569,E2 10779.569} C_VEL
LIN {X 0,Y 388.052,Z 476.03,A -85,B 0,C 180,E1 10786.465,E2 10786.465} C_VEL
LIN {X 0,Y 388.354,Z 476.03,A -85,B 0,C 180,E1 10793.287,E2 10793.287} C_VEL
LIN {X 0,Y 388.761,Z 476.03,A -85,B 0,C 180,E1 10800.003,E2 10800.003} C_VEL
LIN {X 0,Y 388.432,Z 476.03,A -85,B 0,C 180,E1 10806.719,E2 10806.719} C_VEL
LIN {X 0,Y 388.055,Z 476.03,A -85,B 0,C 180,E1 10813.542,E2 10813.542} C_VEL
LIN {X 0,Y 387.817,Z 476.03,A -85,B 0,C 180,E1 10820.574,E2 10820.574} C_VEL
LIN {X 0,Y 387.548,Z 476.03,A -85,B 0,C 180,E1 10827.96,E2 10827.96} C_VEL
LIN {X 0,Y 387.309,Z 476.03,A -85,B 0,C 180,E1 10835.903,E2 10835.903} C_VEL
LIN {X 0,Y 387.236,Z 476.03,A -85,B 0,C 180,E1 10842.021,E2 10842.021} C_VEL
LIN {X 0,Y 387.255,Z 476.03,A -85,B 0,C 180,E1 10848.343,E2 10848.343} C_VEL
LIN {X 0,Y 387.32,Z 476.03,A -85,B 0,C 180,E1 10855.178,E2 10855.178} C_VEL
LIN {X 0,Y 387.519,Z 476.796,A -85,B 0,C 180,E1 10860.028,E2 10860.028} C_VEL
LIN {X 0,Y 405.713,Z 513.4,A -85,B 0,C 180,E1 10863.852,E2 10863.852} C_VEL
LIN {X 0,Y 417.337,Z 544.207,A -85,B 0,C 180,E1 10867.173,E2 10867.173} C_VEL
LIN {X 0,Y 419.055,Z 553.378,A -85,B 0,C 180,E1 10868.086,E2 10868.086} C_VEL
LIN {X 0,Y 413.595,Z 586.608,A -85,B 0,C 180,E1 10870.763,E2 10870.763} C_VEL
LIN {X 0,Y 407.047,Z 619.001,A -85,B 0,C 180,E1 10874.355,E2 10874.355} C_VEL
LIN {X 0,Y 400.548,Z 648.177,A -85,B 0,C 180,E1 10878.83,E2 10878.83} C_VEL
LIN {X 0,Y 395.505,Z 671.294,A -85,B 0,C 180,E1 10883.681,E2 10883.681} C_VEL
LIN {X 0,Y 391.998,Z 689.343,A -85,B 0,C 180,E1 10888.894,E2 10888.894} C_VEL
LIN {X 0,Y 390.022,Z 702.688,A -85,B 0,C 180,E1 10894.453,E2 10894.453} C_VEL
LIN {X 0,Y 389.109,Z 710.963,A -85,B 0,C 180,E1 10900.085,E2 10900.085} C_VEL
LIN {X 0,Y 388.631,Z 713.663,A -85,B 0,C 180,E1 10903.519,E2 10903.519} C_VEL
LIN {X 0,Y 388.474,Z 714.445,A -85,B 0,C 180,E1 10908.169,E2 10908.169} C_VEL
LIN {X 0,Y 388.873,Z 711.961,A -85,B 0,C 180,E1 10912.915,E2 10912.915} C_VEL
LIN {X 0,Y 389.853,Z 704.449,A -85,B 0,C 180,E1 10918.589,E2 10918.589} C_VEL
LIN {X 0,Y 391.693,Z 691.971,A -85,B 0,C 180,E1 10924.161,E2 10924.161} C_VEL
LIN {X 0,Y 394.97,Z 674.478,A -85,B 0,C 180,E1 10929.5,E2 10929.5} C_VEL
LIN {X 0,Y 399.939,Z 651.768,A -85,B 0,C 180,E1 10934.505,E2 10934.505} C_VEL
LIN {X 0,Y 406.241,Z 624.102,A -85,B 0,C 180,E1 10938.981,E2 10938.981} C_VEL
LIN {X 0,Y 412.926,Z 592.325,A -85,B 0,C 180,E1 10942.744,E2 10942.744} C_VEL
LIN {X 0,Y 418.984,Z 557.939,A -85,B 0,C 180,E1 10945.648,E2 10945.648} C_VEL
LIN {X 0,Y 419.433,Z 550.344,A -85,B 0,C 180,E1 10946.256,E2 10946.256} C_VEL
LIN {X 0,Y 408.926,Z 517.689,A -85,B 0,C 180,E1 10949.931,E2 10949.931} C_VEL
LIN {X 0,Y 395.712,Z 491.249,A -85,B 0,C 180,E1 10953.211,E2 10953.211} C_VEL
LIN {X 0,Y 391.054,Z 484.153,A -85,B 0,C 180,E1 10954.269,E2 10954.269} C_VEL
LIN {X 0,Y 389.764,Z 483.191,A -85,B 0,C 180,E1 10954.529,E2 10954.529} C_VEL
LIN {X 0,Y 399.815,Z 520.351,A -85,B 0,C 180,E1 10956.115,E2 10956.115} C_VEL
LIN {X 0,Y 398.536,Z 552.421,A -85,B 0,C 180,E1 10957.826,E2 10957.826} C_VEL
LIN {X 0,Y 396.607,Z 581.752,A -85,B 0,C 180,E1 10960.338,E2 10960.338} C_VEL
LIN {X 0,Y 394.519,Z 606.85,A -85,B 0,C 180,E1 10963.51,E2 10963.51} C_VEL
LIN {X 0,Y 392.905,Z 626.99,A -85,B 0,C 180,E1 10967.195,E2 10967.195} C_VEL
LIN {X 0,Y 391.762,Z 641.483,A -85,B 0,C 180,E1 10971.104,E2 10971.104} C_VEL
LIN {X 0,Y 391.34,Z 651.492,A -85,B 0,C 180,E1 10975.559,E2 10975.559} C_VEL
LIN {X 0,Y 391.345,Z 655.614,A -85,B 0,C 180,E1 10979.997,E2 10979.997} C_VEL
LIN {X 0,Y 391.65,Z 654.14,A -85,B 0,C 180,E1 10984.431,E2 10984.431} C_VEL
LIN {X 0,Y 392.74,Z 646.728,A -85,B 0,C 180,E1 10988.867,E2 10988.867} C_VEL
LIN {X 0,Y 394.308,Z 634.59,A -85,B 0,C 180,E1 10992.751,E2 10992.751} C_VEL
LIN {X 0,Y 396.258,Z 617.49,A -85,B 0,C 180,E1 10996.3,E2 10996.3} C_VEL
LIN {X 0,Y 398.402,Z 595.285,A -85,B 0,C 180,E1 10999.418,E2 10999.418} C_VEL
LIN {X 0,Y 400.309,Z 569.215,A -85,B 0,C 180,E1 11001.897,E2 11001.897} C_VEL
LIN {X 0,Y 401.591,Z 539.072,A -85,B 0,C 180,E1 11003.744,E2 11003.744} C_VEL
LIN {X 0,Y 400.946,Z 514.73,A -85,B 0,C 180,E1 11004.701,E2 11004.701} C_VEL
LIN {X 0,Y 392.463,Z 488.214,A -85,B 0,C 180,E1 11006.125,E2 11006.125} C_VEL
LIN {X 0,Y 387.593,Z 476.03,A -85,B 0,C 180,E1 11007.015,E2 11007.015} C_VEL
LIN {X 0,Y 387.316,Z 476.03,A -85,B 0,C 180,E1 11013.175,E2 11013.175} C_VEL
LIN {X 0,Y 387.305,Z 476.706,A -85,B 0,C 180,E1 11018.913,E2 11018.913} C_VEL
LIN {X 0,Y 390.167,Z 482.067,A -85,B 0,C 180,E1 11019.72,E2 11019.72} C_VEL
LIN {X 0,Y 407.39,Z 511.252,A -85,B 0,C 180,E1 11023.956,E2 11023.956} C_VEL
LIN {X 0,Y 419.587,Z 537.643,A -85,B 0,C 180,E1 11026.916,E2 11026.916} C_VEL
LIN {X 0,Y 423.864,Z 554.143,A -85,B 0,C 180,E1 11028.323,E2 11028.323} C_VEL
LIN {X 0,Y 417.516,Z 597.52,A -85,B 0,C 180,E1 11030.607,E2 11030.607} C_VEL
LIN {X 0,Y 410.638,Z 638.123,A -85,B 0,C 180,E1 11033.682,E2 11033.682} C_VEL
LIN {X 0,Y 404.43,Z 672.876,A -85,B 0,C 180,E1 11037.311,E2 11037.311} C_VEL
LIN {X 0,Y 398.779,Z 703.732,A -85,B 0,C 180,E1 11041.666,E2 11041.666} C_VEL
LIN {X 0,Y 394.248,Z 729.359,A -85,B 0,C 180,E1 11046.519,E2 11046.519} C_VEL
LIN {X 0,Y 391.808,Z 746.088,A -85,B 0,C 180,E1 11050.685,E2 11050.685} C_VEL
LIN {X 0,Y 390.083,Z 749.971,A -85,B 0,C 180,E1 11051.809,E2 11051.809} C_VEL
LIN {X 0,Y 382.415,Z 759.214,A -85,B 0,C 180,E1 11054.938,E2 11054.938} C_VEL
LIN {X 0,Y 382.233,Z 759.968,A -85,B 0,C 180,E1 11055.247,E2 11055.247} C_VEL
LIN {X 0,Y 381.332,Z 771.106,A -85,B 0,C 180,E1 11060.861,E2 11060.861} C_VEL
LIN {X 0,Y 381.029,Z 776.228,A -85,B 0,C 180,E1 11065.441,E2 11065.441} C_VEL
LIN {X 0,Y 381.122,Z 777.988,A -85,B 0,C 180,E1 11070,E2 11070} C_VEL
LIN {X 0,Y 381.103,Z 775.44,A -85,B 0,C 180,E1 11075.674,E2 11075.674} C_VEL
LIN {X 0,Y 381.626,Z 767.55,A -85,B 0,C 180,E1 11081.442,E2 11081.442} C_VEL
LIN {X 0,Y 382.954,Z 753.797,A -85,B 0,C 180,E1 11087.249,E2 11087.249} C_VEL
LIN {X 0,Y 385.943,Z 734.566,A -85,B 0,C 180,E1 11092.779,E2 11092.779} C_VEL
LIN {X 0,Y 390.582,Z 709.221,A -85,B 0,C 180,E1 11098.031,E2 11098.031} C_VEL
LIN {X 0,Y 396.451,Z 679.82,A -85,B 0,C 180,E1 11102.52,E2 11102.52} C_VEL
LIN {X 0,Y 403.275,Z 644.902,A -85,B 0,C 180,E1 11106.421,E2 11106.421} C_VEL
LIN {X 0,Y 410.052,Z 606.204,A -85,B 0,C 180,E1 11109.565,E2 11109.565} C_VEL
LIN {X 0,Y 416.457,Z 566.343,A -85,B 0,C 180,E1 11111.847,E2 11111.847} C_VEL
LIN {X 0,Y 417.33,Z 556.545,A -85,B 0,C 180,E1 11112.343,E2 11112.343} C_VEL
LIN {X 0,Y 408.935,Z 531.935,A -85,B 0,C 180,E1 11114.565,E2 11114.565} C_VEL
LIN {X 0,Y 387.728,Z 492.201,A -85,B 0,C 180,E1 11119.017,E2 11119.017} C_VEL
LIN {X 0,Y 379.491,Z 477.384,A -85,B 0,C 180,E1 11120.798,E2 11120.798} C_VEL
LIN {X 0,Y 379.365,Z 476.03,A -85,B 0,C 180,E1 11121.058,E2 11121.058} C_VEL
LIN {X 0,Y 379.439,Z 476.03,A -85,B 0,C 180,E1 11128.758,E2 11128.758} C_VEL
LIN {X 0,Y 379.661,Z 476.03,A -85,B 0,C 180,E1 11136.527,E2 11136.527} C_VEL
LIN {X 0,Y 380.028,Z 476.03,A -85,B 0,C 180,E1 11143.811,E2 11143.811} C_VEL
LIN {X 0,Y 380.336,Z 476.03,A -85,B 0,C 180,E1 11150.841,E2 11150.841} C_VEL
LIN {X 0,Y 380.763,Z 476.03,A -85,B 0,C 180,E1 11157.725,E2 11157.725} C_VEL
LIN {X 0,Y 380.826,Z 476.03,A -85,B 0,C 180,E1 11162.282,E2 11162.282} C_VEL
LIN {X 0,Y 380.336,Z 476.03,A -85,B 0,C 180,E1 11169.166,E2 11169.166} C_VEL
LIN {X 0,Y 380.011,Z 476.03,A -85,B 0,C 180,E1 11176.197,E2 11176.197} C_VEL
LIN {X 0,Y 379.741,Z 476.03,A -85,B 0,C 180,E1 11183.5,E2 11183.5} C_VEL
LIN {X 0,Y 379.442,Z 476.03,A -85,B 0,C 180,E1 11191.25,E2 11191.25} C_VEL
LIN {X 0,Y 379.298,Z 476.03,A -85,B 0,C 180,E1 11197.025,E2 11197.025} C_VEL
LIN {X 0,Y 379.261,Z 476.03,A -85,B 0,C 180,E1 11204.061,E2 11204.061} C_VEL
LIN {X 0,Y 379.267,Z 476.03,A -85,B 0,C 180,E1 11210.301,E2 11210.301} C_VEL
LIN {X 0,Y 379.434,Z 476.03,A -85,B 0,C 180,E1 11216.929,E2 11216.929} C_VEL
LIN {X 0,Y 379.438,Z 476.402,A -85,B 0,C 180,E1 11218.89,E2 11218.89} C_VEL
LIN {X 0,Y 387.745,Z 492.268,A -85,B 0,C 180,E1 11220.623,E2 11220.623} C_VEL
LIN {X 0,Y 402.23,Z 523.142,A -85,B 0,C 180,E1 11224.004,E2 11224.004} C_VEL
LIN {X 0,Y 412.506,Z 553.039,A -85,B 0,C 180,E1 11227.352,E2 11227.352} C_VEL
LIN {X 0,Y 407.004,Z 587.257,A -85,B 0,C 180,E1 11230.156,E2 11230.156} C_VEL
LIN {X 0,Y 400.391,Z 618.67,A -85,B 0,C 180,E1 11233.665,E2 11233.665} C_VEL
LIN {X 0,Y 393.747,Z 647.502,A -85,B 0,C 180,E1 11238.072,E2 11238.072} C_VEL
LIN {X 0,Y 388.306,Z 670.969,A -85,B 0,C 180,E1 11243.001,E2 11243.001} C_VEL
LIN {X 0,Y 384.496,Z 689.314,A -85,B 0,C 180,E1 11248.308,E2 11248.308} C_VEL
LIN {X 0,Y 382.293,Z 702.891,A -85,B 0,C 180,E1 11253.975,E2 11253.975} C_VEL
LIN {X 0,Y 381.369,Z 710.798,A -85,B 0,C 180,E1 11259.138,E2 11259.138} C_VEL
LIN {X 0,Y 380.73,Z 714.461,A -85,B 0,C 180,E1 11263.805,E2 11263.805} C_VEL
LIN {X 0,Y 380.598,Z 715.048,A -85,B 0,C 180,E1 11268.558,E2 11268.558} C_VEL
LIN {X 0,Y 381.146,Z 711.675,A -85,B 0,C 180,E1 11273.982,E2 11273.982} C_VEL
LIN {X 0,Y 382.161,Z 704.128,A -85,B 0,C 180,E1 11279.351,E2 11279.351} C_VEL
LIN {X 0,Y 384.244,Z 691.106,A -85,B 0,C 180,E1 11285.054,E2 11285.054} C_VEL
LIN {X 0,Y 387.813,Z 673.962,A -85,B 0,C 180,E1 11290.258,E2 11290.258} C_VEL
LIN {X 0,Y 393.061,Z 651.629,A -85,B 0,C 180,E1 11295.205,E2 11295.205} C_VEL
LIN {X 0,Y 399.863,Z 623.438,A -85,B 0,C 180,E1 11299.784,E2 11299.784} C_VEL
LIN {X 0,Y 406.843,Z 591.405,A -85,B 0,C 180,E1 11303.556,E2 11303.556} C_VEL
LIN {X 0,Y 413.062,Z 557.261,A -85,B 0,C 180,E1 11306.433,E2 11306.433} C_VEL
LIN {X 0,Y 411.831,Z 548.937,A -85,B 0,C 180,E1 11307.317,E2 11307.317} C_VEL
LIN {X 0,Y 402.374,Z 519.329,A -85,B 0,C 180,E1 11310.771,E2 11310.771} C_VEL
LIN {X 0,Y 390.809,Z 495.884,A -85,B 0,C 180,E1 11313.826,E2 11313.826} C_VEL
LIN {X 0,Y 386.359,Z 497.188,A -85,B 0,C 180,E1 11314.535,E2 11314.535} C_VEL
LIN {X 0,Y 386.07,Z 497.458,A -85,B 0,C 180,E1 11314.69,E2 11314.69} C_VEL
LIN {X 0,Y 392.334,Z 522.486,A -85,B 0,C 180,E1 11315.813,E2 11315.813} C_VEL
LIN {X 0,Y 390.985,Z 554.086,A -85,B 0,C 180,E1 11317.553,E2 11317.553} C_VEL
LIN {X 0,Y 388.986,Z 583.017,A -85,B 0,C 180,E1 11320.085,E2 11320.085} C_VEL
LIN {X 0,Y 386.824,Z 608.416,A -85,B 0,C 180,E1 11323.36,E2 11323.36} C_VEL
LIN {X 0,Y 385.097,Z 628.98,A -85,B 0,C 180,E1 11327.22,E2 11327.22} C_VEL
LIN {X 0,Y 383.892,Z 644.117,A -85,B 0,C 180,E1 11331.492,E2 11331.492} C_VEL
LIN {X 0,Y 383.575,Z 652.674,A -85,B 0,C 180,E1 11335.469,E2 11335.469} C_VEL
LIN {X 0,Y 383.585,Z 656.968,A -85,B 0,C 180,E1 11339.997,E2 11339.997} C_VEL
LIN {X 0,Y 383.929,Z 655.627,A -85,B 0,C 180,E1 11344.52,E2 11344.52} C_VEL
LIN {X 0,Y 384.933,Z 649.558,A -85,B 0,C 180,E1 11348.478,E2 11348.478} C_VEL
LIN {X 0,Y 386.639,Z 637.309,A -85,B 0,C 180,E1 11352.721,E2 11352.721} C_VEL
LIN {X 0,Y 388.768,Z 620.093,A -85,B 0,C 180,E1 11356.46,E2 11356.46} C_VEL
LIN {X 0,Y 391.077,Z 598.306,A -85,B 0,C 180,E1 11359.65,E2 11359.65} C_VEL
LIN {X 0,Y 393.142,Z 572.564,A -85,B 0,C 180,E1 11362.203,E2 11362.203} C_VEL
LIN {X 0,Y 394.564,Z 541.665,A -85,B 0,C 180,E1 11364.176,E2 11364.176} C_VEL
LIN {X 0,Y 394.133,Z 516.878,A -85,B 0,C 180,E1 11365.186,E2 11365.186} C_VEL
LIN {X 0,Y 386.096,Z 491.448,A -85,B 0,C 180,E1 11366.635,E2 11366.635} C_VEL
LIN {X 0,Y 379.633,Z 476.03,A -85,B 0,C 180,E1 11367.865,E2 11367.865} C_VEL
LIN {X 0,Y 379.38,Z 476.03,A -85,B 0,C 180,E1 11373.962,E2 11373.962} C_VEL
LIN {X 0,Y 379.313,Z 476.7,A -85,B 0,C 180,E1 11377.257,E2 11377.257} C_VEL
LIN {X 0,Y 382.215,Z 482.129,A -85,B 0,C 180,E1 11378.149,E2 11378.149} C_VEL
LIN {X 0,Y 399.763,Z 511.062,A -85,B 0,C 180,E1 11382.781,E2 11382.781} C_VEL
LIN {X 0,Y 413.691,Z 540.977,A -85,B 0,C 180,E1 11386.354,E2 11386.354} C_VEL
LIN {X 0,Y 417.392,Z 557.381,A -85,B 0,C 180,E1 11387.772,E2 11387.772} C_VEL
LIN {X 0,Y 410.622,Z 600.517,A -85,B 0,C 180,E1 11390.157,E2 11390.157} C_VEL
LIN {X 0,Y 403.473,Z 640.493,A -85,B 0,C 180,E1 11393.302,E2 11393.302} C_VEL
LIN {X 0,Y 396.914,Z 675.033,A -85,B 0,C 180,E1 11397.047,E2 11397.047} C_VEL
LIN {X 0,Y 390.79,Z 706.439,A -85,B 0,C 180,E1 11401.694,E2 11401.694} C_VEL
LIN {X 0,Y 386.061,Z 732.346,A -85,B 0,C 180,E1 11406.908,E2 11406.908} C_VEL
LIN {X 0,Y 383.232,Z 751.452,A -85,B 0,C 180,E1 11412.169,E2 11412.169} C_VEL
LIN {X 0,Y 382.233,Z 759.968,A -85,B 0,C 180,E1 11415.247,E2 11415.247} C_VEL
LIN {X 0,Y 380.695,Z 762.852,A -85,B 0,C 180,E1 11416.469,E2 11416.469} C_VEL
LIN {X 0,Y 373.65,Z 769.194,A -85,B 0,C 180,E1 11419.868,E2 11419.868} C_VEL
LIN {X 0,Y 373.513,Z 769.686,A -85,B 0,C 180,E1 11420.196,E2 11420.196} C_VEL
LIN {X 0,Y 373.156,Z 775.562,A -85,B 0,C 180,E1 11425.345,E2 11425.345} C_VEL
LIN {X 0,Y 373.26,Z 777.341,A -85,B 0,C 180,E1 11430,E2 11430} C_VEL
LIN {X 0,Y 373.238,Z 774.986,A -85,B 0,C 180,E1 11435.585,E2 11435.585} C_VEL
LIN {X 0,Y 373.759,Z 766.889,A -85,B 0,C 180,E1 11441.686,E2 11441.686} C_VEL
LIN {X 0,Y 375.223,Z 753.086,A -85,B 0,C 180,E1 11447.616,E2 11447.616} C_VEL
LIN {X 0,Y 378.265,Z 734.202,A -85,B 0,C 180,E1 11453.148,E2 11453.148} C_VEL
LIN {X 0,Y 382.986,Z 709.902,A -85,B 0,C 180,E1 11458.321,E2 11458.321} C_VEL
LIN {X 0,Y 389.221,Z 679.949,A -85,B 0,C 180,E1 11462.998,E2 11462.998} C_VEL
LIN {X 0,Y 395.855,Z 647.261,A -85,B 0,C 180,E1 11466.757,E2 11466.757} C_VEL
LIN {X 0,Y 403.075,Z 608.349,A -85,B 0,C 180,E1 11470.037,E2 11470.037} C_VEL
LIN {X 0,Y 410.052,Z 566.746,A -85,B 0,C 180,E1 11472.481,E2 11472.481} C_VEL
LIN {X 0,Y 410.672,Z 559.044,A -85,B 0,C 180,E1 11472.889,E2 11472.889} C_VEL
LIN {X 0,Y 403.138,Z 536.355,A -85,B 0,C 180,E1 11475.005,E2 11475.005} C_VEL
LIN {X 0,Y 382.686,Z 497.208,A -85,B 0,C 180,E1 11479.548,E2 11479.548} C_VEL
LIN {X 0,Y 371.433,Z 476.668,A -85,B 0,C 180,E1 11482.123,E2 11482.123} C_VEL
LIN {X 0,Y 371.559,Z 476.03,A -85,B 0,C 180,E1 11488.843,E2 11488.843} C_VEL
LIN {X 0,Y 371.685,Z 476.03,A -85,B 0,C 180,E1 11495.966,E2 11495.966} C_VEL
LIN {X 0,Y 372.113,Z 476.03,A -85,B 0,C 180,E1 11503.456,E2 11503.456} C_VEL
LIN {X 0,Y 372.398,Z 476.03,A -85,B 0,C 180,E1 11510.644,E2 11510.644} C_VEL
LIN {X 0,Y 372.853,Z 476.03,A -85,B 0,C 180,E1 11517.676,E2 11517.676} C_VEL
LIN {X 0,Y 372.91,Z 476.03,A -85,B 0,C 180,E1 11522.33,E2 11522.33} C_VEL
LIN {X 0,Y 372.397,Z 476.03,A -85,B 0,C 180,E1 11529.363,E2 11529.363} C_VEL
LIN {X 0,Y 372.089,Z 476.03,A -85,B 0,C 180,E1 11536.552,E2 11536.552} C_VEL
LIN {X 0,Y 371.764,Z 476.03,A -85,B 0,C 180,E1 11544.036,E2 11544.036} C_VEL
LIN {X 0,Y 371.513,Z 476.03,A -85,B 0,C 180,E1 11551.995,E2 11551.995} C_VEL
LIN {X 0,Y 371.337,Z 476.03,A -85,B 0,C 180,E1 11559.221,E2 11559.221} C_VEL
LIN {X 0,Y 371.361,Z 476.03,A -85,B 0,C 180,E1 11566.123,E2 11566.123} C_VEL
LIN {X 0,Y 371.302,Z 476.03,A -85,B 0,C 180,E1 11572.29,E2 11572.29} C_VEL
LIN {X 0,Y 371.5,Z 476.03,A -85,B 0,C 180,E1 11577.674,E2 11577.674} C_VEL
LIN {X 0,Y 374.088,Z 481.888,A -85,B 0,C 180,E1 11578.319,E2 11578.319} C_VEL
LIN {X 0,Y 390.642,Z 514.038,A -85,B 0,C 180,E1 11582.033,E2 11582.033} C_VEL
LIN {X 0,Y 402.619,Z 544.766,A -85,B 0,C 180,E1 11585.565,E2 11585.565} C_VEL
LIN {X 0,Y 405.795,Z 557.777,A -85,B 0,C 180,E1 11587.016,E2 11587.016} C_VEL
LIN {X 0,Y 399.367,Z 593.263,A -85,B 0,C 180,E1 11590.049,E2 11590.049} C_VEL
LIN {X 0,Y 392.423,Z 624.291,A -85,B 0,C 180,E1 11593.756,E2 11593.756} C_VEL
LIN {X 0,Y 385.87,Z 651.119,A -85,B 0,C 180,E1 11598.112,E2 11598.112} C_VEL
LIN {X 0,Y 380.374,Z 673.915,A -85,B 0,C 180,E1 11603.142,E2 11603.142} C_VEL
LIN {X 0,Y 376.403,Z 692.446,A -85,B 0,C 180,E1 11608.848,E2 11608.848} C_VEL
LIN {X 0,Y 374.338,Z 705.214,A -85,B 0,C 180,E1 11614.64,E2 11614.64} C_VEL
LIN {X 0,Y 373.304,Z 712.94,A -85,B 0,C 180,E1 11620.517,E2 11620.517} C_VEL
LIN {X 0,Y 372.715,Z 715.85,A -85,B 0,C 180,E1 11626.521,E2 11626.521} C_VEL
LIN {X 0,Y 372.914,Z 714.508,A -85,B 0,C 180,E1 11631.434,E2 11631.434} C_VEL
LIN {X 0,Y 373.823,Z 708.981,A -85,B 0,C 180,E1 11636.991,E2 11636.991} C_VEL
LIN {X 0,Y 375.595,Z 697.627,A -85,B 0,C 180,E1 11643.117,E2 11643.117} C_VEL
LIN {X 0,Y 379.107,Z 680.532,A -85,B 0,C 180,E1 11649.101,E2 11649.101} C_VEL
LIN {X 0,Y 384.509,Z 658.434,A -85,B 0,C 180,E1 11654.545,E2 11654.545} C_VEL
LIN {X 0,Y 391.201,Z 632.119,A -85,B 0,C 180,E1 11659.255,E2 11659.255} C_VEL
LIN {X 0,Y 398.39,Z 602.112,A -85,B 0,C 180,E1 11663.173,E2 11663.173} C_VEL
LIN {X 0,Y 405.103,Z 569.425,A -85,B 0,C 180,E1 11666.272,E2 11666.272} C_VEL
LIN {X 0,Y 406.952,Z 557.224,A -85,B 0,C 180,E1 11667.227,E2 11667.227} C_VEL
LIN {X 0,Y 397.624,Z 525.276,A -85,B 0,C 180,E1 11671.115,E2 11671.115} C_VEL
LIN {X 0,Y 388.813,Z 505.88,A -85,B 0,C 180,E1 11673.7,E2 11673.7} C_VEL
LIN {X 0,Y 383.987,Z 510.302,A -85,B 0,C 180,E1 11674.293,E2 11674.293} C_VEL
LIN {X 0,Y 381.761,Z 509.954,A -85,B 0,C 180,E1 11674.793,E2 11674.793} C_VEL
LIN {X 0,Y 384.8,Z 525.223,A -85,B 0,C 180,E1 11675.537,E2 11675.537} C_VEL
LIN {X 0,Y 383.378,Z 556.336,A -85,B 0,C 180,E1 11677.326,E2 11677.326} C_VEL
LIN {X 0,Y 381.274,Z 585.487,A -85,B 0,C 180,E1 11679.968,E2 11679.968} C_VEL
LIN {X 0,Y 379.026,Z 610.907,A -85,B 0,C 180,E1 11683.359,E2 11683.359} C_VEL
LIN {X 0,Y 377.287,Z 630.945,A -85,B 0,C 180,E1 11687.246,E2 11687.246} C_VEL
LIN {X 0,Y 376.159,Z 645.089,A -85,B 0,C 180,E1 11691.315,E2 11691.315} C_VEL
LIN {X 0,Y 375.777,Z 653.85,A -85,B 0,C 180,E1 11695.375,E2 11695.375} C_VEL
LIN {X 0,Y 375.818,Z 658.32,A -85,B 0,C 180,E1 11699.996,E2 11699.996} C_VEL
LIN {X 0,Y 376.224,Z 657.128,A -85,B 0,C 180,E1 11704.613,E2 11704.613} C_VEL
LIN {X 0,Y 377.478,Z 649.966,A -85,B 0,C 180,E1 11709.228,E2 11709.228} C_VEL
LIN {X 0,Y 379.43,Z 636.859,A -85,B 0,C 180,E1 11713.554,E2 11713.554} C_VEL
LIN {X 0,Y 381.664,Z 619.876,A -85,B 0,C 180,E1 11717.149,E2 11717.149} C_VEL
LIN {X 0,Y 384.229,Z 596.575,A -85,B 0,C 180,E1 11720.466,E2 11720.466} C_VEL
LIN {X 0,Y 386.348,Z 569.324,A -85,B 0,C 180,E1 11723.067,E2 11723.067} C_VEL
LIN {X 0,Y 387.703,Z 537.723,A -85,B 0,C 180,E1 11724.954,E2 11724.954} C_VEL
LIN {X 0,Y 387.259,Z 518.553,A -85,B 0,C 180,E1 11725.73,E2 11725.73} C_VEL
LIN {X 0,Y 379.623,Z 494.274,A -85,B 0,C 180,E1 11727.208,E2 11727.208} C_VEL
LIN {X 0,Y 371.562,Z 476.03,A -85,B 0,C 180,E1 11728.917,E2 11728.917} C_VEL
LIN {X 0,Y 371.355,Z 476.288,A -85,B 0,C 180,E1 11735.409,E2 11735.409} C_VEL
LIN {X 0,Y 373.587,Z 481.52,A -85,B 0,C 180,E1 11736.223,E2 11736.223} C_VEL
LIN {X 0,Y 377.003,Z 486.754,A -85,B 0,C 180,E1 11737.283,E2 11737.283} C_VEL
LIN {X 0,Y 390.108,Z 507.818,A -85,B 0,C 180,E1 11741.001,E2 11741.001} C_VEL
LIN {X 0,Y 404.96,Z 537.33,A -85,B 0,C 180,E1 11744.984,E2 11744.984} C_VEL
LIN {X 0,Y 411.134,Z 557.782,A -85,B 0,C 180,E1 11747.046,E2 11747.046} C_VEL
LIN {X 0,Y 403.707,Z 603.607,A -85,B 0,C 180,E1 11749.686,E2 11749.686} C_VEL
LIN {X 0,Y 395.936,Z 645.107,A -85,B 0,C 180,E1 11753.124,E2 11753.124} C_VEL
LIN {X 0,Y 388.832,Z 679.826,A -85,B 0,C 180,E1 11757.13,E2 11757.13} C_VEL
LIN {X 0,Y 382.882,Z 708.773,A -85,B 0,C 180,E1 11761.67,E2 11761.67} C_VEL
LIN {X 0,Y 378.073,Z 734.236,A -85,B 0,C 180,E1 11767.07,E2 11767.07} C_VEL
LIN {X 0,Y 375.24,Z 752.462,A -85,B 0,C 180,E1 11772.384,E2 11772.384} C_VEL
LIN {X 0,Y 373.702,Z 766.508,A -85,B 0,C 180,E1 11778.311,E2 11778.311} C_VEL
LIN {X 0,Y 373.513,Z 769.686,A -85,B 0,C 180,E1 11780.196,E2 11780.196} C_VEL
LIN {X 0,Y 370.834,Z 772.309,A -85,B 0,C 180,E1 11782.134,E2 11782.134} C_VEL
LIN {X 0,Y 365.26,Z 775.006,A -85,B 0,C 180,E1 11785.435,E2 11785.435} C_VEL
LIN {X 0,Y 365.384,Z 776.692,A -85,B 0,C 180,E1 11790,E2 11790} C_VEL
LIN {X 0,Y 365.3,Z 775.053,A -85,B 0,C 180,E1 11794.755,E2 11794.755} C_VEL
LIN {X 0,Y 365.771,Z 768.258,A -85,B 0,C 180,E1 11800.735,E2 11800.735} C_VEL
LIN {X 0,Y 366.977,Z 755.62,A -85,B 0,C 180,E1 11806.787,E2 11806.787} C_VEL
LIN {X 0,Y 369.845,Z 737.886,A -85,B 0,C 180,E1 11812.474,E2 11812.474} C_VEL
LIN {X 0,Y 374.725,Z 713.583,A -85,B 0,C 180,E1 11818.035,E2 11818.035} C_VEL
LIN {X 0,Y 381.129,Z 684.077,A -85,B 0,C 180,E1 11822.94,E2 11822.94} C_VEL
LIN {X 0,Y 388.293,Z 650.612,A -85,B 0,C 180,E1 11827,E2 11827} C_VEL
LIN {X 0,Y 395.777,Z 611.811,A -85,B 0,C 180,E1 11830.407,E2 11830.407} C_VEL
LIN {X 0,Y 403.125,Z 570.036,A -85,B 0,C 180,E1 11832.988,E2 11832.988} C_VEL
LIN {X 0,Y 403.967,Z 561.313,A -85,B 0,C 180,E1 11833.472,E2 11833.472} C_VEL
LIN {X 0,Y 397.309,Z 540.697,A -85,B 0,C 180,E1 11835.466,E2 11835.466} C_VEL
LIN {X 0,Y 377.777,Z 502.525,A -85,B 0,C 180,E1 11840.028,E2 11840.028} C_VEL
LIN {X 0,Y 363.539,Z 477.436,A -85,B 0,C 180,E1 11843.422,E2 11843.422} C_VEL
LIN {X 0,Y 363.39,Z 476.03,A -85,B 0,C 180,E1 11843.739,E2 11843.739} C_VEL
LIN {X 0,Y 363.632,Z 476.03,A -85,B 0,C 180,E1 11850.975,E2 11850.975} C_VEL
LIN {X 0,Y 363.824,Z 476.03,A -85,B 0,C 180,E1 11858.009,E2 11858.009} C_VEL
LIN {X 0,Y 364.22,Z 476.03,A -85,B 0,C 180,E1 11865.561,E2 11865.561} C_VEL
LIN {X 0,Y 364.593,Z 476.03,A -85,B 0,C 180,E1 11872.847,E2 11872.847} C_VEL
LIN {X 0,Y 365.056,Z 476.03,A -85,B 0,C 180,E1 11880.004,E2 11880.004} C_VEL
LIN {X 0,Y 364.683,Z 476.03,A -85,B 0,C 180,E1 11887.158,E2 11887.158} C_VEL
LIN {X 0,Y 364.216,Z 476.03,A -85,B 0,C 180,E1 11894.447,E2 11894.447} C_VEL
LIN {X 0,Y 363.891,Z 476.03,A -85,B 0,C 180,E1 11901.994,E2 11901.994} C_VEL
LIN {X 0,Y 363.638,Z 476.03,A -85,B 0,C 180,E1 11909.979,E2 11909.979} C_VEL
LIN {X 0,Y 363.423,Z 476.03,A -85,B 0,C 180,E1 11917.666,E2 11917.666} C_VEL
LIN {X 0,Y 363.407,Z 476.03,A -85,B 0,C 180,E1 11925.097,E2 11925.097} C_VEL
LIN {X 0,Y 363.412,Z 476.03,A -85,B 0,C 180,E1 11932.337,E2 11932.337} C_VEL
LIN {X 0,Y 363.59,Z 476.128,A -85,B 0,C 180,E1 11936.467,E2 11936.467} C_VEL
LIN {X 0,Y 366.029,Z 481.697,A -85,B 0,C 180,E1 11937.089,E2 11937.089} C_VEL
LIN {X 0,Y 383.47,Z 515.051,A -85,B 0,C 180,E1 11941.142,E2 11941.142} C_VEL
LIN {X 0,Y 395.363,Z 545.42,A -85,B 0,C 180,E1 11944.756,E2 11944.756} C_VEL
LIN {X 0,Y 399.072,Z 560.787,A -85,B 0,C 180,E1 11946.52,E2 11946.52} C_VEL
LIN {X 0,Y 392.214,Z 596.339,A -85,B 0,C 180,E1 11949.67,E2 11949.67} C_VEL
LIN {X 0,Y 385.117,Z 626.833,A -85,B 0,C 180,E1 11953.439,E2 11953.439} C_VEL
LIN {X 0,Y 378.354,Z 653.278,A -85,B 0,C 180,E1 11957.872,E2 11957.872} C_VEL
LIN {X 0,Y 372.699,Z 675.718,A -85,B 0,C 180,E1 11963,E2 11963} C_VEL
LIN {X 0,Y 368.595,Z 693.975,A -85,B 0,C 180,E1 11968.824,E2 11968.824} C_VEL
LIN {X 0,Y 366.487,Z 706.461,A -85,B 0,C 180,E1 11974.74,E2 11974.74} C_VEL
LIN {X 0,Y 365.418,Z 713.922,A -85,B 0,C 180,E1 11980.747,E2 11980.747} C_VEL
LIN {X 0,Y 364.828,Z 716.554,A -85,B 0,C 180,E1 11986.889,E2 11986.889} C_VEL
LIN {X 0,Y 365.082,Z 714.905,A -85,B 0,C 180,E1 11991.917,E2 11991.917} C_VEL
LIN {X 0,Y 365.998,Z 709.839,A -85,B 0,C 180,E1 11997.07,E2 11997.07} C_VEL
LIN {X 0,Y 367.665,Z 699.804,A -85,B 0,C 180,E1 12002.799,E2 12002.799} C_VEL
LIN {X 0,Y 371.138,Z 683.53,A -85,B 0,C 180,E1 12008.884,E2 12008.884} C_VEL
LIN {X 0,Y 376.42,Z 662.935,A -85,B 0,C 180,E1 12014.287,E2 12014.287} C_VEL
LIN {X 0,Y 383.466,Z 636.741,A -85,B 0,C 180,E1 12019.273,E2 12019.273} C_VEL
LIN {X 0,Y 391.188,Z 606.568,A -85,B 0,C 180,E1 12023.447,E2 12023.447} C_VEL
LIN {X 0,Y 398.445,Z 573.535,A -85,B 0,C 180,E1 12026.722,E2 12026.722} C_VEL
LIN {X 0,Y 400.668,Z 560.368,A -85,B 0,C 180,E1 12027.777,E2 12027.777} C_VEL
LIN {X 0,Y 392.495,Z 530.555,A -85,B 0,C 180,E1 12031.538,E2 12031.538} C_VEL
LIN {X 0,Y 386.114,Z 516.478,A -85,B 0,C 180,E1 12033.56,E2 12033.56} C_VEL
LIN {X 0,Y 382.556,Z 519.264,A -85,B 0,C 180,E1 12034.011,E2 12034.011} C_VEL
LIN {X 0,Y 379.309,Z 522.098,A -85,B 0,C 180,E1 12034.406,E2 12034.406} C_VEL
LIN {X 0,Y 376.8,Z 521.554,A -85,B 0,C 180,E1 12034.947,E2 12034.947} C_VEL
LIN {X 0,Y 376.187,Z 551.71,A -85,B 0,C 180,E1 12036.601,E2 12036.601} C_VEL
LIN {X 0,Y 374.104,Z 581.143,A -85,B 0,C 180,E1 12039.102,E2 12039.102} C_VEL
LIN {X 0,Y 371.844,Z 607.155,A -85,B 0,C 180,E1 12042.369,E2 12042.369} C_VEL
LIN {X 0,Y 369.974,Z 627.705,A -85,B 0,C 180,E1 12046.085,E2 12046.085} C_VEL
LIN {X 0,Y 368.533,Z 643.983,A -85,B 0,C 180,E1 12050.418,E2 12050.418} C_VEL
LIN {X 0,Y 367.971,Z 654.06,A -85,B 0,C 180,E1 12054.685,E2 12054.685} C_VEL
LIN {X 0,Y 367.907,Z 658.07,A -85,B 0,C 180,E1 12057.638,E2 12057.638} C_VEL
LIN {X 0,Y 368.165,Z 659.882,A -85,B 0,C 180,E1 12062.353,E2 12062.353} C_VEL
LIN {X 0,Y 369.146,Z 655.906,A -85,B 0,C 180,E1 12067.064,E2 12067.064} C_VEL
LIN {X 0,Y 370.604,Z 646.869,A -85,B 0,C 180,E1 12071.323,E2 12071.323} C_VEL
LIN {X 0,Y 372.899,Z 632.658,A -85,B 0,C 180,E1 12075.298,E2 12075.298} C_VEL
LIN {X 0,Y 375.351,Z 613.782,A -85,B 0,C 180,E1 12078.822,E2 12078.822} C_VEL
LIN {X 0,Y 378.1,Z 588.673,A -85,B 0,C 180,E1 12081.973,E2 12081.973} C_VEL
LIN {X 0,Y 380.161,Z 559.121,A -85,B 0,C 180,E1 12084.413,E2 12084.413} C_VEL
LIN {X 0,Y 381.202,Z 527.826,A -85,B 0,C 180,E1 12085.974,E2 12085.974} C_VEL
LIN {X 0,Y 378.751,Z 512.999,A -85,B 0,C 180,E1 12086.704,E2 12086.704} C_VEL
LIN {X 0,Y 370.213,Z 490.268,A -85,B 0,C 180,E1 12088.448,E2 12088.448} C_VEL
LIN {X 0,Y 363.606,Z 476.03,A -85,B 0,C 180,E1 12089.973,E2 12089.973} C_VEL
LIN {X 0,Y 363.422,Z 476.206,A -85,B 0,C 180,E1 12093.388,E2 12093.388} C_VEL
LIN {X 0,Y 365.673,Z 481.547,A -85,B 0,C 180,E1 12094.323,E2 12094.323} C_VEL
LIN {X 0,Y 368.116,Z 484.971,A -85,B 0,C 180,E1 12095.151,E2 12095.151} C_VEL
LIN {X 0,Y 382.255,Z 507.426,A -85,B 0,C 180,E1 12099.543,E2 12099.543} C_VEL
LIN {X 0,Y 396.992,Z 536.146,A -85,B 0,C 180,E1 12103.775,E2 12103.775} C_VEL
LIN {X 0,Y 403.44,Z 554.537,A -85,B 0,C 180,E1 12105.861,E2 12105.861} C_VEL
LIN {X 0,Y 404.602,Z 562.63,A -85,B 0,C 180,E1 12106.57,E2 12106.57} C_VEL
LIN {X 0,Y 397.195,Z 604.665,A -85,B 0,C 180,E1 12109.065,E2 12109.065} C_VEL
LIN {X 0,Y 389.323,Z 644.822,A -85,B 0,C 180,E1 12112.447,E2 12112.447} C_VEL
LIN {X 0,Y 381.937,Z 679.078,A -85,B 0,C 180,E1 12116.459,E2 12116.459} C_VEL
LIN {X 0,Y 375.329,Z 709.499,A -85,B 0,C 180,E1 12121.349,E2 12121.349} C_VEL
LIN {X 0,Y 370.383,Z 734.088,A -85,B 0,C 180,E1 12126.732,E2 12126.732} C_VEL
LIN {X 0,Y 367.427,Z 752.266,A -85,B 0,C 180,E1 12132.191,E2 12132.191} C_VEL
LIN {X 0,Y 365.861,Z 765.814,A -85,B 0,C 180,E1 12138.057,E2 12138.057} C_VEL
LIN {X 0,Y 365.333,Z 773.896,A -85,B 0,C 180,E1 12144.009,E2 12144.009} C_VEL
LIN {X 0,Y 365.26,Z 775.006,A -85,B 0,C 180,E1 12145.435,E2 12145.435} C_VEL
LIN {X 0,Y 362.729,Z 775.946,A -85,B 0,C 180,E1 12147.452,E2 12147.452} C_VEL
LIN {X 0,Y 357.447,Z 775.903,A -85,B 0,C 180,E1 12150.853,E2 12150.853} C_VEL
LIN {X 0,Y 357.459,Z 773.421,A -85,B 0,C 180,E1 12156.135,E2 12156.135} C_VEL
LIN {X 0,Y 358.059,Z 765.531,A -85,B 0,C 180,E1 12162.206,E2 12162.206} C_VEL
LIN {X 0,Y 359.611,Z 752.422,A -85,B 0,C 180,E1 12168.1,E2 12168.1} C_VEL
LIN {X 0,Y 362.895,Z 733.745,A -85,B 0,C 180,E1 12173.859,E2 12173.859} C_VEL
LIN {X 0,Y 368.132,Z 709.488,A -85,B 0,C 180,E1 12179.236,E2 12179.236} C_VEL
LIN {X 0,Y 374.9,Z 679.88,A -85,B 0,C 180,E1 12184.054,E2 12184.054} C_VEL
LIN {X 0,Y 382.525,Z 645.51,A -85,B 0,C 180,E1 12188.116,E2 12188.116} C_VEL
LIN {X 0,Y 390.263,Z 606.525,A -85,B 0,C 180,E1 12191.442,E2 12191.442} C_VEL
LIN {X 0,Y 397.427,Z 563.967,A -85,B 0,C 180,E1 12194.02,E2 12194.02} C_VEL
LIN {X 0,Y 391.534,Z 545.208,A -85,B 0,C 180,E1 12195.895,E2 12195.895} C_VEL
LIN {X 0,Y 372.665,Z 507.546,A -85,B 0,C 180,E1 12200.544,E2 12200.544} C_VEL
LIN {X 0,Y 355.584,Z 477.198,A -85,B 0,C 180,E1 12204.853,E2 12204.853} C_VEL
LIN {X 0,Y 355.498,Z 476.03,A -85,B 0,C 180,E1 12205.027,E2 12205.027} C_VEL
LIN {X 0,Y 355.723,Z 476.03,A -85,B 0,C 180,E1 12212.088,E2 12212.088} C_VEL
LIN {X 0,Y 356.04,Z 476.03,A -85,B 0,C 180,E1 12220.116,E2 12220.116} C_VEL
LIN {X 0,Y 356.422,Z 476.03,A -85,B 0,C 180,E1 12227.741,E2 12227.741} C_VEL
LIN {X 0,Y 356.919,Z 476.03,A -85,B 0,C 180,E1 12235.137,E2 12235.137} C_VEL
LIN {X 0,Y 357.105,Z 476.03,A -85,B 0,C 180,E1 12242.434,E2 12242.434} C_VEL
LIN {X 0,Y 356.517,Z 476.03,A -85,B 0,C 180,E1 12249.784,E2 12249.784} C_VEL
LIN {X 0,Y 356.207,Z 476.03,A -85,B 0,C 180,E1 12257.313,E2 12257.313} C_VEL
LIN {X 0,Y 355.808,Z 476.03,A -85,B 0,C 180,E1 12265.187,E2 12265.187} C_VEL
LIN {X 0,Y 355.544,Z 476.03,A -85,B 0,C 180,E1 12271.602,E2 12271.602} C_VEL
LIN {X 0,Y 355.48,Z 476.03,A -85,B 0,C 180,E1 12276.608,E2 12276.608} C_VEL
LIN {X 0,Y 355.393,Z 476.03,A -85,B 0,C 180,E1 12283.593,E2 12283.593} C_VEL
LIN {X 0,Y 355.436,Z 476.03,A -85,B 0,C 180,E1 12290.285,E2 12290.285} C_VEL
LIN {X 0,Y 355.513,Z 476.03,A -85,B 0,C 180,E1 12295.107,E2 12295.107} C_VEL
LIN {X 0,Y 358.138,Z 481.82,A -85,B 0,C 180,E1 12295.821,E2 12295.821} C_VEL
LIN {X 0,Y 375.851,Z 515.134,A -85,B 0,C 180,E1 12300.096,E2 12300.096} C_VEL
LIN {X 0,Y 388.313,Z 546.651,A -85,B 0,C 180,E1 12303.983,E2 12303.983} C_VEL
LIN {X 0,Y 392.51,Z 562.924,A -85,B 0,C 180,E1 12305.948,E2 12305.948} C_VEL
LIN {X 0,Y 385.375,Z 598.139,A -85,B 0,C 180,E1 12309.142,E2 12309.142} C_VEL
LIN {X 0,Y 378.284,Z 627.469,A -85,B 0,C 180,E1 12312.831,E2 12312.831} C_VEL
LIN {X 0,Y 371.219,Z 653.951,A -85,B 0,C 180,E1 12317.336,E2 12317.336} C_VEL
LIN {X 0,Y 365.269,Z 676.436,A -85,B 0,C 180,E1 12322.558,E2 12322.558} C_VEL
LIN {X 0,Y 361.109,Z 693.883,A -85,B 0,C 180,E1 12328.198,E2 12328.198} C_VEL
LIN {X 0,Y 358.752,Z 706.636,A -85,B 0,C 180,E1 12334.236,E2 12334.236} C_VEL
LIN {X 0,Y 357.697,Z 713.732,A -85,B 0,C 180,E1 12339.749,E2 12339.749} C_VEL
LIN {X 0,Y 357.034,Z 716.855,A -85,B 0,C 180,E1 12344.741,E2 12344.741} C_VEL
LIN {X 0,Y 357.099,Z 716.154,A -85,B 0,C 180,E1 12351.123,E2 12351.123} C_VEL
LIN {X 0,Y 358.204,Z 710.337,A -85,B 0,C 180,E1 12357.419,E2 12357.419} C_VEL
LIN {X 0,Y 360.24,Z 699.252,A -85,B 0,C 180,E1 12363.715,E2 12363.715} C_VEL
LIN {X 0,Y 364.11,Z 682.86,A -85,B 0,C 180,E1 12369.781,E2 12369.781} C_VEL
LIN {X 0,Y 369.74,Z 662.3,A -85,B 0,C 180,E1 12375.17,E2 12375.17} C_VEL
LIN {X 0,Y 377.133,Z 636.299,A -85,B 0,C 180,E1 12380.132,E2 12380.132} C_VEL
LIN {X 0,Y 385.34,Z 605.502,A -85,B 0,C 180,E1 12384.368,E2 12384.368} C_VEL
LIN {X 0,Y 392.894,Z 572.14,A -85,B 0,C 180,E1 12387.651,E2 12387.651} C_VEL
LIN {X 0,Y 394.193,Z 562.344,A -85,B 0,C 180,E1 12388.507,E2 12388.507} C_VEL
LIN {X 0,Y 386.57,Z 533.57,A -85,B 0,C 180,E1 12392.28,E2 12392.28} C_VEL
LIN {X 0,Y 383.319,Z 526.379,A -85,B 0,C 180,E1 12393.378,E2 12393.378} C_VEL
LIN {X 0,Y 377.423,Z 530.647,A -85,B 0,C 180,E1 12394.132,E2 12394.132} C_VEL
LIN {X 0,Y 371.989,Z 536.259,A -85,B 0,C 180,E1 12394.696,E2 12394.696} C_VEL
LIN {X 0,Y 369.597,Z 536.135,A -85,B 0,C 180,E1 12395.25,E2 12395.25} C_VEL
LIN {X 0,Y 367.676,Z 567.902,A -85,B 0,C 180,E1 12397.442,E2 12397.442} C_VEL
LIN {X 0,Y 365.295,Z 596.459,A -85,B 0,C 180,E1 12400.475,E2 12400.475} C_VEL
LIN {X 0,Y 363.05,Z 619.737,A -85,B 0,C 180,E1 12404.07,E2 12404.07} C_VEL
LIN {X 0,Y 361.354,Z 638.213,A -85,B 0,C 180,E1 12408.21,E2 12408.21} C_VEL
LIN {X 0,Y 360.357,Z 651.509,A -85,B 0,C 180,E1 12412.755,E2 12412.755} C_VEL
LIN {X 0,Y 360.133,Z 659.322,A -85,B 0,C 180,E1 12417.587,E2 12417.587} C_VEL
LIN {X 0,Y 360.419,Z 661.334,A -85,B 0,C 180,E1 12422.404,E2 12422.404} C_VEL
LIN {X 0,Y 361.496,Z 657.498,A -85,B 0,C 180,E1 12427.214,E2 12427.214} C_VEL
LIN {X 0,Y 363.026,Z 648.879,A -85,B 0,C 180,E1 12431.463,E2 12431.463} C_VEL
LIN {X 0,Y 365.519,Z 634.553,A -85,B 0,C 180,E1 12435.615,E2 12435.615} C_VEL
LIN {X 0,Y 368.16,Z 615.816,A -85,B 0,C 180,E1 12439.204,E2 12439.204} C_VEL
LIN {X 0,Y 370.962,Z 591.658,A -85,B 0,C 180,E1 12442.346,E2 12442.346} C_VEL
LIN {X 0,Y 373.202,Z 563.147,A -85,B 0,C 180,E1 12444.807,E2 12444.807} C_VEL
LIN {X 0,Y 374.544,Z 530.973,A -85,B 0,C 180,E1 12446.519,E2 12446.519} C_VEL
LIN {X 0,Y 373.07,Z 518.337,A -85,B 0,C 180,E1 12447.127,E2 12447.127} C_VEL
LIN {X 0,Y 365.178,Z 495.681,A -85,B 0,C 180,E1 12448.891,E2 12448.891} C_VEL
LIN {X 0,Y 356.76,Z 480.205,A -85,B 0,C 180,E1 12450.845,E2 12450.845} C_VEL
LIN {X 0,Y 355.611,Z 476.94,A -85,B 0,C 180,E1 12451.21,E2 12451.21} C_VEL
LIN {X 0,Y 358.421,Z 482.139,A -85,B 0,C 180,E1 12452.417,E2 12452.417} C_VEL
LIN {X 0,Y 369.009,Z 498.509,A -85,B 0,C 180,E1 12456.229,E2 12456.229} C_VEL
LIN {X 0,Y 383.675,Z 523.929,A -85,B 0,C 180,E1 12460.836,E2 12460.836} C_VEL
LIN {X 0,Y 395.913,Z 551.593,A -85,B 0,C 180,E1 12464.637,E2 12464.637} C_VEL
LIN {X 0,Y 398.441,Z 564.424,A -85,B 0,C 180,E1 12465.895,E2 12465.895} C_VEL
LIN {X 0,Y 390.466,Z 607.77,A -85,B 0,C 180,E1 12468.575,E2 12468.575} C_VEL
LIN {X 0,Y 382.195,Z 647.339,A -85,B 0,C 180,E1 12472.031,E2 12472.031} C_VEL
LIN {X 0,Y 374.478,Z 681.075,A -85,B 0,C 180,E1 12476.147,E2 12476.147} C_VEL
LIN {X 0,Y 367.711,Z 710.516,A -85,B 0,C 180,E1 12481.064,E2 12481.064} C_VEL
LIN {X 0,Y 362.438,Z 735.476,A -85,B 0,C 180,E1 12486.771,E2 12486.771} C_VEL
LIN {X 0,Y 359.225,Z 754.365,A -85,B 0,C 180,E1 12492.839,E2 12492.839} C_VEL
LIN {X 0,Y 357.868,Z 767.228,A -85,B 0,C 180,E1 12499.024,E2 12499.024} C_VEL
LIN {X 0,Y 357.407,Z 774.246,A -85,B 0,C 180,E1 12505.139,E2 12505.139} C_VEL
LIN {X 0,Y 357.447,Z 775.903,A -85,B 0,C 180,E1 12510.853,E2 12510.853} C_VEL
LIN {X 0,Y 354.897,Z 775.267,A -85,B 0,C 180,E1 12512.914,E2 12512.914} C_VEL
LIN {X 0,Y 349.573,Z 772.665,A -85,B 0,C 180,E1 12516.366,E2 12516.366} C_VEL
LIN {X 0,Y 350.214,Z 764.833,A -85,B 0,C 180,E1 12522.484,E2 12522.484} C_VEL
LIN {X 0,Y 352.028,Z 750.61,A -85,B 0,C 180,E1 12528.895,E2 12528.895} C_VEL
LIN {X 0,Y 355.742,Z 731.235,A -85,B 0,C 180,E1 12534.82,E2 12534.82} C_VEL
LIN {X 0,Y 361.712,Z 705.384,A -85,B 0,C 180,E1 12540.468,E2 12540.468} C_VEL
LIN {X 0,Y 368.897,Z 675.126,A -85,B 0,C 180,E1 12545.252,E2 12545.252} C_VEL
LIN {X 0,Y 376.486,Z 641.932,A -85,B 0,C 180,E1 12549.089,E2 12549.089} C_VEL
LIN {X 0,Y 384.427,Z 602.979,A -85,B 0,C 180,E1 12552.365,E2 12552.365} C_VEL
LIN {X 0,Y 390.803,Z 566.33,A -85,B 0,C 180,E1 12554.605,E2 12554.605} C_VEL
LIN {X 0,Y 385.487,Z 549.141,A -85,B 0,C 180,E1 12556.393,E2 12556.393} C_VEL
LIN {X 0,Y 367.18,Z 511.833,A -85,B 0,C 180,E1 12561.161,E2 12561.161} C_VEL
LIN {X 0,Y 349.725,Z 481.405,A -85,B 0,C 180,E1 12565.756,E2 12565.756} C_VEL
LIN {X 0,Y 347.639,Z 476.03,A -85,B 0,C 180,E1 12566.565,E2 12566.565} C_VEL
LIN {X 0,Y 347.81,Z 476.03,A -85,B 0,C 180,E1 12574.2,E2 12574.2} C_VEL
LIN {X 0,Y 348.262,Z 476.03,A -85,B 0,C 180,E1 12582.287,E2 12582.287} C_VEL
LIN {X 0,Y 348.586,Z 476.03,A -85,B 0,C 180,E1 12589.999,E2 12589.999} C_VEL
LIN {X 0,Y 349.148,Z 476.03,A -85,B 0,C 180,E1 12597.519,E2 12597.519} C_VEL
LIN {X 0,Y 349.012,Z 476.03,A -85,B 0,C 180,E1 12603.801,E2 12603.801} C_VEL
LIN {X 0,Y 348.579,Z 476.03,A -85,B 0,C 180,E1 12610.009,E2 12610.009} C_VEL
LIN {X 0,Y 348.244,Z 476.03,A -85,B 0,C 180,E1 12617.722,E2 12617.722} C_VEL
LIN {X 0,Y 347.864,Z 476.03,A -85,B 0,C 180,E1 12625.804,E2 12625.804} C_VEL
LIN {X 0,Y 347.662,Z 476.03,A -85,B 0,C 180,E1 12631.51,E2 12631.51} C_VEL
LIN {X 0,Y 347.433,Z 476.03,A -85,B 0,C 180,E1 12638.332,E2 12638.332} C_VEL
LIN {X 0,Y 347.422,Z 476.03,A -85,B 0,C 180,E1 12645.79,E2 12645.79} C_VEL
LIN {X 0,Y 347.582,Z 476.118,A -85,B 0,C 180,E1 12653.708,E2 12653.708} C_VEL
LIN {X 0,Y 350.047,Z 481.723,A -85,B 0,C 180,E1 12654.421,E2 12654.421} C_VEL
LIN {X 0,Y 368.406,Z 515.337,A -85,B 0,C 180,E1 12659.026,E2 12659.026} C_VEL
LIN {X 0,Y 380.682,Z 546.046,A -85,B 0,C 180,E1 12662.945,E2 12662.945} C_VEL
LIN {X 0,Y 385.849,Z 565.714,A -85,B 0,C 180,E1 12665.413,E2 12665.413} C_VEL
LIN {X 0,Y 378.562,Z 599.884,A -85,B 0,C 180,E1 12668.595,E2 12668.595} C_VEL
LIN {X 0,Y 370.992,Z 629.944,A -85,B 0,C 180,E1 12672.483,E2 12672.483} C_VEL
LIN {X 0,Y 363.312,Z 657.493,A -85,B 0,C 180,E1 12677.362,E2 12677.362} C_VEL
LIN {X 0,Y 357.313,Z 679.292,A -85,B 0,C 180,E1 12682.697,E2 12682.697} C_VEL
LIN {X 0,Y 352.963,Z 696.861,A -85,B 0,C 180,E1 12688.771,E2 12688.771} C_VEL
LIN {X 0,Y 350.761,Z 708.771,A -85,B 0,C 180,E1 12694.953,E2 12694.953} C_VEL
LIN {X 0,Y 349.775,Z 714.704,A -85,B 0,C 180,E1 12699.972,E2 12699.972} C_VEL
LIN {X 0,Y 349.136,Z 717.597,A -85,B 0,C 180,E1 12705.083,E2 12705.083} C_VEL
LIN {X 0,Y 349.159,Z 717.167,A -85,B 0,C 180,E1 12710.299,E2 12710.299} C_VEL
LIN {X 0,Y 350.22,Z 712.058,A -85,B 0,C 180,E1 12716.786,E2 12716.786} C_VEL
LIN {X 0,Y 352.247,Z 701.563,A -85,B 0,C 180,E1 12723.335,E2 12723.335} C_VEL
LIN {X 0,Y 356.152,Z 685.714,A -85,B 0,C 180,E1 12729.621,E2 12729.621} C_VEL
LIN {X 0,Y 362.106,Z 665.127,A -85,B 0,C 180,E1 12735.304,E2 12735.304} C_VEL
LIN {X 0,Y 369.636,Z 640.102,A -85,B 0,C 180,E1 12740.305,E2 12740.305} C_VEL
LIN {X 0,Y 378.12,Z 610.13,A -85,B 0,C 180,E1 12744.656,E2 12744.656} C_VEL
LIN {X 0,Y 386.141,Z 577.132,A -85,B 0,C 180,E1 12748.069,E2 12748.069} C_VEL
LIN {X 0,Y 387.97,Z 565.006,A -85,B 0,C 180,E1 12749.159,E2 12749.159} C_VEL
LIN {X 0,Y 381.269,Z 538.143,A -85,B 0,C 180,E1 12752.824,E2 12752.824} C_VEL
LIN {X 0,Y 379.073,Z 536.733,A -85,B 0,C 180,E1 12753.325,E2 12753.325} C_VEL
LIN {X 0,Y 371.898,Z 543.139,A -85,B 0,C 180,E1 12754.109,E2 12754.109} C_VEL
LIN {X 0,Y 365.158,Z 549.088,A -85,B 0,C 180,E1 12754.847,E2 12754.847} C_VEL
LIN {X 0,Y 361.342,Z 549.683,A -85,B 0,C 180,E1 12755.637,E2 12755.637} C_VEL
LIN {X 0,Y 359.159,Z 580.576,A -85,B 0,C 180,E1 12758.225,E2 12758.225} C_VEL
LIN {X 0,Y 356.666,Z 607.375,A -85,B 0,C 180,E1 12761.592,E2 12761.592} C_VEL
LIN {X 0,Y 354.613,Z 628.744,A -85,B 0,C 180,E1 12765.469,E2 12765.469} C_VEL
LIN {X 0,Y 353.146,Z 644.182,A -85,B 0,C 180,E1 12769.498,E2 12769.498} C_VEL
LIN {X 0,Y 352.434,Z 655.119,A -85,B 0,C 180,E1 12773.831,E2 12773.831} C_VEL
LIN {X 0,Y 352.369,Z 660.578,A -85,B 0,C 180,E1 12777.534,E2 12777.534} C_VEL
LIN {X 0,Y 352.663,Z 662.784,A -85,B 0,C 180,E1 12782.457,E2 12782.457} C_VEL
LIN {X 0,Y 353.827,Z 659.142,A -85,B 0,C 180,E1 12787.372,E2 12787.372} C_VEL
LIN {X 0,Y 355.422,Z 651.119,A -85,B 0,C 180,E1 12791.53,E2 12791.53} C_VEL
LIN {X 0,Y 358.158,Z 636.481,A -85,B 0,C 180,E1 12795.944,E2 12795.944} C_VEL
LIN {X 0,Y 361.007,Z 617.947,A -85,B 0,C 180,E1 12799.599,E2 12799.599} C_VEL
LIN {X 0,Y 363.954,Z 594.629,A -85,B 0,C 180,E1 12802.739,E2 12802.739} C_VEL
LIN {X 0,Y 366.455,Z 565.84,A -85,B 0,C 180,E1 12805.33,E2 12805.33} C_VEL
LIN {X 0,Y 367.966,Z 534.77,A -85,B 0,C 180,E1 12807.072,E2 12807.072} C_VEL
LIN {X 0,Y 367.105,Z 522.608,A -85,B 0,C 180,E1 12807.642,E2 12807.642} C_VEL
LIN {X 0,Y 360.118,Z 501.106,A -85,B 0,C 180,E1 12809.37,E2 12809.37} C_VEL
LIN {X 0,Y 353.182,Z 486.878,A -85,B 0,C 180,E1 12811.236,E2 12811.236} C_VEL
LIN {X 0,Y 357.178,Z 492.131,A -85,B 0,C 180,E1 12812.817,E2 12812.817} C_VEL
LIN {X 0,Y 370.718,Z 513.978,A -85,B 0,C 180,E1 12817.665,E2 12817.665} C_VEL
LIN {X 0,Y 384.8,Z 541.942,A -85,B 0,C 180,E1 12822.257,E2 12822.257} C_VEL
LIN {X 0,Y 391.505,Z 561.054,A -85,B 0,C 180,E1 12824.69,E2 12824.69} C_VEL
LIN {X 0,Y 391.95,Z 568.182,A -85,B 0,C 180,E1 12825.308,E2 12825.308} C_VEL
LIN {X 0,Y 383.575,Z 611.119,A -85,B 0,C 180,E1 12828.074,E2 12828.074} C_VEL
LIN {X 0,Y 374.86,Z 650.693,A -85,B 0,C 180,E1 12831.686,E2 12831.686} C_VEL
LIN {X 0,Y 366.884,Z 683.583,A -85,B 0,C 180,E1 12835.897,E2 12835.897} C_VEL
LIN {X 0,Y 359.773,Z 712.942,A -85,B 0,C 180,E1 12841.054,E2 12841.054} C_VEL
LIN {X 0,Y 354.494,Z 736.766,A -85,B 0,C 180,E1 12846.807,E2 12846.807} C_VEL
LIN {X 0,Y 351.486,Z 753.684,A -85,B 0,C 180,E1 12852.449,E2 12852.449} C_VEL
LIN {X 0,Y 350.011,Z 766.56,A -85,B 0,C 180,E1 12858.774,E2 12858.774} C_VEL
LIN {X 0,Y 349.535,Z 773.591,A -85,B 0,C 180,E1 12865.029,E2 12865.029} C_VEL
LIN {X 0,Y 349.568,Z 775.258,A -85,B 0,C 180,E1 12870.837,E2 12870.837} C_VEL
LIN {X 0,Y 349.573,Z 772.665,A -85,B 0,C 180,E1 12876.366,E2 12876.366} C_VEL
LIN {X 0,Y 347.172,Z 770.469,A -85,B 0,C 180,E1 12878.458,E2 12878.458} C_VEL
LIN {X 0,Y 342.281,Z 766.052,A -85,B 0,C 180,E1 12881.581,E2 12881.581} C_VEL
LIN {X 0,Y 342.249,Z 765.469,A -85,B 0,C 180,E1 12881.938,E2 12881.938} C_VEL
LIN {X 0,Y 343.728,Z 753.368,A -85,B 0,C 180,E1 12887.959,E2 12887.959} C_VEL
LIN {X 0,Y 347.135,Z 735.627,A -85,B 0,C 180,E1 12893.949,E2 12893.949} C_VEL
LIN {X 0,Y 352.593,Z 712.182,A -85,B 0,C 180,E1 12899.593,E2 12899.593} C_VEL
LIN {X 0,Y 359.521,Z 684.465,A -85,B 0,C 180,E1 12904.492,E2 12904.492} C_VEL
LIN {X 0,Y 367.586,Z 651.184,A -85,B 0,C 180,E1 12908.77,E2 12908.77} C_VEL
LIN {X 0,Y 375.958,Z 612.744,A -85,B 0,C 180,E1 12912.325,E2 12912.325} C_VEL
LIN {X 0,Y 384.33,Z 569.098,A -85,B 0,C 180,E1 12915.164,E2 12915.164} C_VEL
LIN {X 0,Y 379.293,Z 552.69,A -85,B 0,C 180,E1 12916.943,E2 12916.943} C_VEL
LIN {X 0,Y 360.715,Z 514.17,A -85,B 0,C 180,E1 12922.041,E2 12922.041} C_VEL
LIN {X 0,Y 341.803,Z 481.383,A -85,B 0,C 180,E1 12927.312,E2 12927.312} C_VEL
LIN {X 0,Y 339.719,Z 476.03,A -85,B 0,C 180,E1 12928.163,E2 12928.163} C_VEL
LIN {X 0,Y 339.929,Z 476.03,A -85,B 0,C 180,E1 12936.373,E2 12936.373} C_VEL
LIN {X 0,Y 340.393,Z 476.03,A -85,B 0,C 180,E1 12944.526,E2 12944.526} C_VEL
LIN {X 0,Y 340.805,Z 476.03,A -85,B 0,C 180,E1 12952.345,E2 12952.345} C_VEL
LIN {X 0,Y 341.376,Z 476.03,A -85,B 0,C 180,E1 12960.004,E2 12960.004} C_VEL
LIN {X 0,Y 340.867,Z 476.03,A -85,B 0,C 180,E1 12967.661,E2 12967.661} C_VEL
LIN {X 0,Y 340.383,Z 476.03,A -85,B 0,C 180,E1 12975.483,E2 12975.483} C_VEL
LIN {X 0,Y 340.163,Z 476.03,A -85,B 0,C 180,E1 12980.863,E2 12980.863} C_VEL
LIN {X 0,Y 339.808,Z 476.03,A -85,B 0,C 180,E1 12989.352,E2 12989.352} C_VEL
LIN {X 0,Y 339.484,Z 476.03,A -85,B 0,C 180,E1 12996.602,E2 12996.602} C_VEL
LIN {X 0,Y 339.507,Z 476.03,A -85,B 0,C 180,E1 13001.989,E2 13001.989} C_VEL
LIN {X 0,Y 339.513,Z 476.03,A -85,B 0,C 180,E1 13009.302,E2 13009.302} C_VEL
LIN {X 0,Y 339.559,Z 476.03,A -85,B 0,C 180,E1 13012.146,E2 13012.146} C_VEL
LIN {X 0,Y 341.996,Z 481.702,A -85,B 0,C 180,E1 13012.932,E2 13012.932} C_VEL
LIN {X 0,Y 359.43,Z 512.54,A -85,B 0,C 180,E1 13017.503,E2 13017.503} C_VEL
LIN {X 0,Y 371.784,Z 541.91,A -85,B 0,C 180,E1 13021.411,E2 13021.411} C_VEL
LIN {X 0,Y 379.3,Z 567.829,A -85,B 0,C 180,E1 13024.813,E2 13024.813} C_VEL
LIN {X 0,Y 371.791,Z 601.597,A -85,B 0,C 180,E1 13028.028,E2 13028.028} C_VEL
LIN {X 0,Y 364.217,Z 630.521,A -85,B 0,C 180,E1 13031.833,E2 13031.833} C_VEL
LIN {X 0,Y 356.639,Z 656.672,A -85,B 0,C 180,E1 13036.497,E2 13036.497} C_VEL
LIN {X 0,Y 349.913,Z 679.959,A -85,B 0,C 180,E1 13042.229,E2 13042.229} C_VEL
LIN {X 0,Y 345.132,Z 698.245,A -85,B 0,C 180,E1 13048.744,E2 13048.744} C_VEL
LIN {X 0,Y 342.868,Z 709.906,A -85,B 0,C 180,E1 13055.067,E2 13055.067} C_VEL
LIN {X 0,Y 341.859,Z 715.669,A -85,B 0,C 180,E1 13060.205,E2 13060.205} C_VEL
LIN {X 0,Y 341.216,Z 718.297,A -85,B 0,C 180,E1 13065.441,E2 13065.441} C_VEL
LIN {X 0,Y 341.376,Z 717.474,A -85,B 0,C 180,E1 13071.343,E2 13071.343} C_VEL
LIN {X 0,Y 342.623,Z 711.735,A -85,B 0,C 180,E1 13077.891,E2 13077.891} C_VEL
LIN {X 0,Y 344.757,Z 701.745,A -85,B 0,C 180,E1 13083.995,E2 13083.995} C_VEL
LIN {X 0,Y 349.193,Z 685.105,A -85,B 0,C 180,E1 13090.573,E2 13090.573} C_VEL
LIN {X 0,Y 355.717,Z 664.082,A -85,B 0,C 180,E1 13096.354,E2 13096.354} C_VEL
LIN {X 0,Y 364.14,Z 637.525,A -85,B 0,C 180,E1 13101.593,E2 13101.593} C_VEL
LIN {X 0,Y 373.055,Z 606.853,A -85,B 0,C 180,E1 13105.906,E2 13105.906} C_VEL
LIN {X 0,Y 381.255,Z 573.592,A -85,B 0,C 180,E1 13109.247,E2 13109.247} C_VEL
LIN {X 0,Y 381.643,Z 566.99,A -85,B 0,C 180,E1 13109.941,E2 13109.941} C_VEL
LIN {X 0,Y 377.005,Z 546.348,A -85,B 0,C 180,E1 13112.848,E2 13112.848} C_VEL
LIN {X 0,Y 365.26,Z 555.6,A -85,B 0,C 180,E1 13114.146,E2 13114.146} C_VEL
LIN {X 0,Y 360.719,Z 557.737,A -85,B 0,C 180,E1 13114.835,E2 13114.835} C_VEL
LIN {X 0,Y 358.674,Z 559.72,A -85,B 0,C 180,E1 13115.028,E2 13115.028} C_VEL
LIN {X 0,Y 353.188,Z 561.312,A -85,B 0,C 180,E1 13116.049,E2 13116.049} C_VEL
LIN {X 0,Y 350.804,Z 590.227,A -85,B 0,C 180,E1 13118.875,E2 13118.875} C_VEL
LIN {X 0,Y 348.408,Z 614.333,A -85,B 0,C 180,E1 13122.287,E2 13122.287} C_VEL
LIN {X 0,Y 346.372,Z 634.696,A -85,B 0,C 180,E1 13126.408,E2 13126.408} C_VEL
LIN {X 0,Y 345.068,Z 649.906,A -85,B 0,C 180,E1 13130.963,E2 13130.963} C_VEL
LIN {X 0,Y 344.604,Z 658.433,A -85,B 0,C 180,E1 13134.955,E2 13134.955} C_VEL
LIN {X 0,Y 344.745,Z 663.739,A -85,B 0,C 180,E1 13139.996,E2 13139.996} C_VEL
LIN {X 0,Y 345.355,Z 663.282,A -85,B 0,C 180,E1 13145.026,E2 13145.026} C_VEL
LIN {X 0,Y 347.09,Z 656.77,A -85,B 0,C 180,E1 13150.044,E2 13150.044} C_VEL
LIN {X 0,Y 349.709,Z 644.358,A -85,B 0,C 180,E1 13154.731,E2 13154.731} C_VEL
LIN {X 0,Y 352.898,Z 626.364,A -85,B 0,C 180,E1 13158.917,E2 13158.917} C_VEL
LIN {X 0,Y 356.288,Z 603.247,A -85,B 0,C 180,E1 13162.481,E2 13162.481} C_VEL
LIN {X 0,Y 359.112,Z 576.464,A -85,B 0,C 180,E1 13165.265,E2 13165.265} C_VEL
LIN {X 0,Y 361.256,Z 544.201,A -85,B 0,C 180,E1 13167.391,E2 13167.391} C_VEL
LIN {X 0,Y 361.028,Z 525.7,A -85,B 0,C 180,E1 13168.27,E2 13168.27} C_VEL
LIN {X 0,Y 354.644,Z 505.146,A -85,B 0,C 180,E1 13170.015,E2 13170.015} C_VEL
LIN {X 0,Y 350.552,Z 496.113,A -85,B 0,C 180,E1 13171.212,E2 13171.212} C_VEL
LIN {X 0,Y 353.051,Z 497.204,A -85,B 0,C 180,E1 13172.047,E2 13172.047} C_VEL
LIN {X 0,Y 366.932,Z 520.967,A -85,B 0,C 180,E1 13177.39,E2 13177.39} C_VEL
LIN {X 0,Y 379.713,Z 547.219,A -85,B 0,C 180,E1 13181.819,E2 13181.819} C_VEL
LIN {X 0,Y 385.716,Z 565.05,A -85,B 0,C 180,E1 13184.165,E2 13184.165} C_VEL
LIN {X 0,Y 385.752,Z 570.926,A -85,B 0,C 180,E1 13184.648,E2 13184.648} C_VEL
LIN {X 0,Y 376.926,Z 613.556,A -85,B 0,C 180,E1 13187.493,E2 13187.493} C_VEL
LIN {X 0,Y 368.329,Z 650.955,A -85,B 0,C 180,E1 13190.99,E2 13190.99} C_VEL
LIN {X 0,Y 359.873,Z 684.031,A -85,B 0,C 180,E1 13195.322,E2 13195.322} C_VEL
LIN {X 0,Y 352.597,Z 712.327,A -85,B 0,C 180,E1 13200.407,E2 13200.407} C_VEL
LIN {X 0,Y 346.859,Z 736.67,A -85,B 0,C 180,E1 13206.428,E2 13206.428} C_VEL
LIN {X 0,Y 343.474,Z 754.607,A -85,B 0,C 180,E1 13212.689,E2 13212.689} C_VEL
LIN {X 0,Y 342.145,Z 765.898,A -85,B 0,C 180,E1 13218.513,E2 13218.513} C_VEL
LIN {X 0,Y 341.67,Z 772.949,A -85,B 0,C 180,E1 13224.915,E2 13224.915} C_VEL
LIN {X 0,Y 341.783,Z 774.742,A -85,B 0,C 180,E1 13230,E2 13230} C_VEL
LIN {X 0,Y 341.67,Z 773.082,A -85,B 0,C 180,E1 13235.084,E2 13235.084} C_VEL
LIN {X 0,Y 342.184,Z 766.198,A -85,B 0,C 180,E1 13241.485,E2 13241.485} C_VEL
LIN {X 0,Y 342.249,Z 765.469,A -85,B 0,C 180,E1 13241.938,E2 13241.938} C_VEL
LIN {X 0,Y 340.088,Z 761.851,A -85,B 0,C 180,E1 13244.025,E2 13244.025} C_VEL
LIN {X 0,Y 335.58,Z 755.497,A -85,B 0,C 180,E1 13247.13,E2 13247.13} C_VEL
LIN {X 0,Y 335.623,Z 754.712,A -85,B 0,C 180,E1 13247.483,E2 13247.483} C_VEL
LIN {X 0,Y 339.04,Z 737.457,A -85,B 0,C 180,E1 13253.698,E2 13253.698} C_VEL
LIN {X 0,Y 344.614,Z 714.245,A -85,B 0,C 180,E1 13259.622,E2 13259.622} C_VEL
LIN {X 0,Y 351.915,Z 686.174,A -85,B 0,C 180,E1 13264.789,E2 13264.789} C_VEL
LIN {X 0,Y 360.11,Z 654.083,A -85,B 0,C 180,E1 13269.1,E2 13269.1} C_VEL
LIN {X 0,Y 368.878,Z 615.293,A -85,B 0,C 180,E1 13272.817,E2 13272.817} C_VEL
LIN {X 0,Y 377.54,Z 570.431,A -85,B 0,C 180,E1 13275.871,E2 13275.871} C_VEL
LIN {X 0,Y 372.258,Z 554.206,A -85,B 0,C 180,E1 13277.75,E2 13277.75} C_VEL
LIN {X 0,Y 353.294,Z 514.747,A -85,B 0,C 180,E1 13283.234,E2 13283.234} C_VEL
LIN {X 0,Y 334.381,Z 481.798,A -85,B 0,C 180,E1 13288.859,E2 13288.859} C_VEL
LIN {X 0,Y 331.825,Z 476.03,A -85,B 0,C 180,E1 13289.879,E2 13289.879} C_VEL
LIN {X 0,Y 331.967,Z 476.03,A -85,B 0,C 180,E1 13295.811,E2 13295.811} C_VEL
LIN {X 0,Y 332.431,Z 476.03,A -85,B 0,C 180,E1 13304.146,E2 13304.146} C_VEL
LIN {X 0,Y 332.883,Z 476.03,A -85,B 0,C 180,E1 13312.162,E2 13312.162} C_VEL
LIN {X 0,Y 333.474,Z 476.03,A -85,B 0,C 180,E1 13320.004,E2 13320.004} C_VEL
LIN {X 0,Y 332.935,Z 476.03,A -85,B 0,C 180,E1 13327.845,E2 13327.845} C_VEL
LIN {X 0,Y 332.421,Z 476.03,A -85,B 0,C 180,E1 13335.863,E2 13335.863} C_VEL
LIN {X 0,Y 332.168,Z 476.03,A -85,B 0,C 180,E1 13341.389,E2 13341.389} C_VEL
LIN {X 0,Y 331.854,Z 476.03,A -85,B 0,C 180,E1 13349.901,E2 13349.901} C_VEL
LIN {X 0,Y 331.604,Z 476.03,A -85,B 0,C 180,E1 13356.414,E2 13356.414} C_VEL
LIN {X 0,Y 331.537,Z 476.03,A -85,B 0,C 180,E1 13363.241,E2 13363.241} C_VEL
LIN {X 0,Y 331.581,Z 476.538,A -85,B 0,C 180,E1 13370.541,E2 13370.541} C_VEL
LIN {X 0,Y 334.279,Z 481.937,A -85,B 0,C 180,E1 13371.413,E2 13371.413} C_VEL
LIN {X 0,Y 351.375,Z 511.865,A -85,B 0,C 180,E1 13376.151,E2 13376.151} C_VEL
LIN {X 0,Y 364.293,Z 541.55,A -85,B 0,C 180,E1 13380.298,E2 13380.298} C_VEL
LIN {X 0,Y 372.778,Z 569.919,A -85,B 0,C 180,E1 13384.196,E2 13384.196} C_VEL
LIN {X 0,Y 365.054,Z 603.261,A -85,B 0,C 180,E1 13387.44,E2 13387.44} C_VEL
LIN {X 0,Y 356.977,Z 632.919,A -85,B 0,C 180,E1 13391.452,E2 13391.452} C_VEL
LIN {X 0,Y 348.7,Z 660.16,A -85,B 0,C 180,E1 13396.504,E2 13396.504} C_VEL
LIN {X 0,Y 341.913,Z 682.624,A -85,B 0,C 180,E1 13402.366,E2 13402.366} C_VEL
LIN {X 0,Y 337.301,Z 699.628,A -85,B 0,C 180,E1 13408.714,E2 13408.714} C_VEL
LIN {X 0,Y 334.985,Z 711.023,A -85,B 0,C 180,E1 13415.187,E2 13415.187} C_VEL
LIN {X 0,Y 333.923,Z 716.627,A -85,B 0,C 180,E1 13420.45,E2 13420.45} C_VEL
LIN {X 0,Y 333.284,Z 719.128,A -85,B 0,C 180,E1 13427.44,E2 13427.44} C_VEL
LIN {X 0,Y 333.933,Z 716.467,A -85,B 0,C 180,E1 13434.085,E2 13434.085} C_VEL
LIN {X 0,Y 335.693,Z 708.393,A -85,B 0,C 180,E1 13441.02,E2 13441.02} C_VEL
LIN {X 0,Y 338.781,Z 695.923,A -85,B 0,C 180,E1 13447.381,E2 13447.381} C_VEL
LIN {X 0,Y 344.642,Z 677.286,A -85,B 0,C 180,E1 13453.789,E2 13453.789} C_VEL
LIN {X 0,Y 352.821,Z 653.027,A -85,B 0,C 180,E1 13459.611,E2 13459.611} C_VEL
LIN {X 0,Y 361.861,Z 625.165,A -85,B 0,C 180,E1 13464.382,E2 13464.382} C_VEL
LIN {X 0,Y 370.995,Z 593.421,A -85,B 0,C 180,E1 13468.294,E2 13468.294} C_VEL
LIN {X 0,Y 375.902,Z 571.803,A -85,B 0,C 180,E1 13470.343,E2 13470.343} C_VEL
LIN {X 0,Y 373.321,Z 557.693,A -85,B 0,C 180,E1 13472.378,E2 13472.378} C_VEL
LIN {X 0,Y 371.645,Z 556.799,A -85,B 0,C 180,E1 13472.785,E2 13472.785} C_VEL
LIN {X 0,Y 363.271,Z 562.846,A -85,B 0,C 180,E1 13473.705,E2 13473.705} C_VEL
LIN {X 0,Y 350.361,Z 570.611,A -85,B 0,C 180,E1 13475.454,E2 13475.454} C_VEL
LIN {X 0,Y 345.223,Z 572.288,A -85,B 0,C 180,E1 13476.406,E2 13476.406} C_VEL
LIN {X 0,Y 344.612,Z 575.502,A -85,B 0,C 180,E1 13476.864,E2 13476.864} C_VEL
LIN {X 0,Y 342.017,Z 602.919,A -85,B 0,C 180,E1 13480.101,E2 13480.101} C_VEL
LIN {X 0,Y 339.59,Z 626.58,A -85,B 0,C 180,E1 13484.152,E2 13484.152} C_VEL
LIN {X 0,Y 337.755,Z 644.709,A -85,B 0,C 180,E1 13488.686,E2 13488.686} C_VEL
LIN {X 0,Y 336.892,Z 657.222,A -85,B 0,C 180,E1 13493.545,E2 13493.545} C_VEL
LIN {X 0,Y 336.818,Z 664.265,A -85,B 0,C 180,E1 13498.708,E2 13498.708} C_VEL
LIN {X 0,Y 337.153,Z 665.715,A -85,B 0,C 180,E1 13502.57,E2 13502.57} C_VEL
LIN {X 0,Y 338.536,Z 662.471,A -85,B 0,C 180,E1 13507.706,E2 13507.706} C_VEL
LIN {X 0,Y 340.527,Z 654.239,A -85,B 0,C 180,E1 13512.287,E2 13512.287} C_VEL
LIN {X 0,Y 343.55,Z 640.605,A -85,B 0,C 180,E1 13516.642,E2 13516.642} C_VEL
LIN {X 0,Y 346.787,Z 622.578,A -85,B 0,C 180,E1 13520.438,E2 13520.438} C_VEL
LIN {X 0,Y 350.381,Z 598.396,A -85,B 0,C 180,E1 13523.884,E2 13523.884} C_VEL
LIN {X 0,Y 353.421,Z 569.508,A -85,B 0,C 180,E1 13526.611,E2 13526.611} C_VEL
LIN {X 0,Y 355.291,Z 538.444,A -85,B 0,C 180,E1 13528.468,E2 13528.468} C_VEL
LIN {X 0,Y 354.623,Z 526.394,A -85,B 0,C 180,E1 13529.1,E2 13529.1} C_VEL
LIN {X 0,Y 348.441,Z 507.185,A -85,B 0,C 180,E1 13530.95,E2 13530.95} C_VEL
LIN {X 0,Y 348.185,Z 505.278,A -85,B 0,C 180,E1 13531.321,E2 13531.321} C_VEL
LIN {X 0,Y 350,Z 504.757,A -85,B 0,C 180,E1 13531.812,E2 13531.812} C_VEL
LIN {X 0,Y 362.59,Z 526.707,A -85,B 0,C 180,E1 13536.883,E2 13536.883} C_VEL
LIN {X 0,Y 374.781,Z 552.809,A -85,B 0,C 180,E1 13541.41,E2 13541.41} C_VEL
LIN {X 0,Y 379.993,Z 569.311,A -85,B 0,C 180,E1 13543.655,E2 13543.655} C_VEL
LIN {X 0,Y 370.299,Z 616.42,A -85,B 0,C 180,E1 13546.908,E2 13546.908} C_VEL
LIN {X 0,Y 361.36,Z 653.121,A -85,B 0,C 180,E1 13550.478,E2 13550.478} C_VEL
LIN {X 0,Y 352.458,Z 685.951,A -85,B 0,C 180,E1 13554.953,E2 13554.953} C_VEL
LIN {X 0,Y 344.631,Z 714.692,A -85,B 0,C 180,E1 13560.378,E2 13560.378} C_VEL
LIN {X 0,Y 339.02,Z 737.456,A -85,B 0,C 180,E1 13566.299,E2 13566.299} C_VEL
LIN {X 0,Y 335.488,Z 755.459,A -85,B 0,C 180,E1 13572.941,E2 13572.941} C_VEL
LIN {X 0,Y 334.103,Z 767.119,A -85,B 0,C 180,E1 13579.555,E2 13579.555} C_VEL
LIN {X 0,Y 333.795,Z 772.302,A -85,B 0,C 180,E1 13584.794,E2 13584.794} C_VEL
LIN {X 0,Y 333.907,Z 774.089,A -85,B 0,C 180,E1 13590,E2 13590} C_VEL
LIN {X 0,Y 333.829,Z 771.472,A -85,B 0,C 180,E1 13596.51,E2 13596.51} C_VEL
LIN {X 0,Y 334.53,Z 763.395,A -85,B 0,C 180,E1 13603.079,E2 13603.079} C_VEL
LIN {X 0,Y 335.623,Z 754.712,A -85,B 0,C 180,E1 13607.483,E2 13607.483} C_VEL
LIN {X 0,Y 334.955,Z 751.522,A -85,B 0,C 180,E1 13608.872,E2 13608.872} C_VEL
LIN {X 0,Y 330.413,Z 741.71,A -85,B 0,C 180,E1 13612.617,E2 13612.617} C_VEL
LIN {X 0,Y 330.553,Z 740.685,A -85,B 0,C 180,E1 13612.955,E2 13612.955} C_VEL
LIN {X 0,Y 335.97,Z 718.75,A -85,B 0,C 180,E1 13619.055,E2 13619.055} C_VEL
LIN {X 0,Y 343.457,Z 690.997,A -85,B 0,C 180,E1 13624.582,E2 13624.582} C_VEL
LIN {X 0,Y 351.994,Z 659.125,A -85,B 0,C 180,E1 13629.169,E2 13629.169} C_VEL
LIN {X 0,Y 360.977,Z 621.34,A -85,B 0,C 180,E1 13633.045,E2 13633.045} C_VEL
LIN {X 0,Y 370.378,Z 577.864,A -85,B 0,C 180,E1 13636.156,E2 13636.156} C_VEL
LIN {X 0,Y 370.749,Z 571.598,A -85,B 0,C 180,E1 13636.621,E2 13636.621} C_VEL
LIN {X 0,Y 363.721,Z 552.463,A -85,B 0,C 180,E1 13639.04,E2 13639.04} C_VEL
LIN {X 0,Y 345.243,Z 514.31,A -85,B 0,C 180,E1 13644.673,E2 13644.673} C_VEL
LIN {X 0,Y 329.145,Z 486.496,A -85,B 0,C 180,E1 13649.722,E2 13649.722} C_VEL
LIN {X 0,Y 325.321,Z 480.568,A -85,B 0,C 180,E1 13651.001,E2 13651.001} C_VEL
LIN {X 0,Y 323.899,Z 476.03,A -85,B 0,C 180,E1 13651.798,E2 13651.798} C_VEL
LIN {X 0,Y 324.193,Z 476.03,A -85,B 0,C 180,E1 13659.079,E2 13659.079} C_VEL
LIN {X 0,Y 324.635,Z 476.03,A -85,B 0,C 180,E1 13666.52,E2 13666.52} C_VEL
LIN {X 0,Y 325.206,Z 476.03,A -85,B 0,C 180,E1 13674.662,E2 13674.662} C_VEL
LIN {X 0,Y 325.588,Z 476.03,A -85,B 0,C 180,E1 13680.004,E2 13680.004} C_VEL
LIN {X 0,Y 324.989,Z 476.03,A -85,B 0,C 180,E1 13688.038,E2 13688.038} C_VEL
LIN {X 0,Y 324.489,Z 476.03,A -85,B 0,C 180,E1 13696.261,E2 13696.261} C_VEL
LIN {X 0,Y 324.195,Z 476.03,A -85,B 0,C 180,E1 13701.942,E2 13701.942} C_VEL
LIN {X 0,Y 323.933,Z 476.03,A -85,B 0,C 180,E1 13707.869,E2 13707.869} C_VEL
LIN {X 0,Y 323.68,Z 476.03,A -85,B 0,C 180,E1 13714.15,E2 13714.15} C_VEL
LIN {X 0,Y 323.518,Z 476.03,A -85,B 0,C 180,E1 13721.512,E2 13721.512} C_VEL
LIN {X 0,Y 323.546,Z 476.339,A -85,B 0,C 180,E1 13728.728,E2 13728.728} C_VEL
LIN {X 0,Y 325.962,Z 481.689,A -85,B 0,C 180,E1 13729.602,E2 13729.602} C_VEL
LIN {X 0,Y 341.433,Z 507.394,A -85,B 0,C 180,E1 13734.166,E2 13734.166} C_VEL
LIN {X 0,Y 354.501,Z 535.402,A -85,B 0,C 180,E1 13738.302,E2 13738.302} C_VEL
LIN {X 0,Y 364.208,Z 564.393,A -85,B 0,C 180,E1 13742.452,E2 13742.452} C_VEL
LIN {X 0,Y 365.851,Z 574.022,A -85,B 0,C 180,E1 13743.733,E2 13743.733} C_VEL
LIN {X 0,Y 357.738,Z 607.28,A -85,B 0,C 180,E1 13747.117,E2 13747.117} C_VEL
LIN {X 0,Y 349.153,Z 637.163,A -85,B 0,C 180,E1 13751.348,E2 13751.348} C_VEL
LIN {X 0,Y 340.772,Z 663.438,A -85,B 0,C 180,E1 13756.511,E2 13756.511} C_VEL
LIN {X 0,Y 334.223,Z 684.253,A -85,B 0,C 180,E1 13762.189,E2 13762.189} C_VEL
LIN {X 0,Y 329.471,Z 700.983,A -85,B 0,C 180,E1 13768.684,E2 13768.684} C_VEL
LIN {X 0,Y 327.107,Z 712.139,A -85,B 0,C 180,E1 13775.312,E2 13775.312} C_VEL
LIN {X 0,Y 326,Z 717.51,A -85,B 0,C 180,E1 13780.707,E2 13780.707} C_VEL
LIN {X 0,Y 325.447,Z 719.697,A -85,B 0,C 180,E1 13786.21,E2 13786.21} C_VEL
LIN {X 0,Y 325.668,Z 718.672,A -85,B 0,C 180,E1 13791.836,E2 13791.836} C_VEL
LIN {X 0,Y 327.045,Z 713.185,A -85,B 0,C 180,E1 13798.4,E2 13798.4} C_VEL
LIN {X 0,Y 329.771,Z 702.336,A -85,B 0,C 180,E1 13805.252,E2 13805.252} C_VEL
LIN {X 0,Y 334.976,Z 685.655,A -85,B 0,C 180,E1 13812.029,E2 13812.029} C_VEL
LIN {X 0,Y 342.642,Z 663.894,A -85,B 0,C 180,E1 13818.139,E2 13818.139} C_VEL
LIN {X 0,Y 352.087,Z 636.797,A -85,B 0,C 180,E1 13823.497,E2 13823.497} C_VEL
LIN {X 0,Y 361.255,Z 607.855,A -85,B 0,C 180,E1 13827.61,E2 13827.61} C_VEL
LIN {X 0,Y 369.836,Z 574.404,A -85,B 0,C 180,E1 13831.077,E2 13831.077} C_VEL
LIN {X 0,Y 368.713,Z 567.207,A -85,B 0,C 180,E1 13832.151,E2 13832.151} C_VEL
LIN {X 0,Y 367.773,Z 566.568,A -85,B 0,C 180,E1 13832.407,E2 13832.407} C_VEL
LIN {X 0,Y 345.501,Z 578.96,A -85,B 0,C 180,E1 13835.342,E2 13835.342} C_VEL
LIN {X 0,Y 339.337,Z 582.047,A -85,B 0,C 180,E1 13836.321,E2 13836.321} C_VEL
LIN {X 0,Y 336.537,Z 582.083,A -85,B 0,C 180,E1 13837.095,E2 13837.095} C_VEL
LIN {X 0,Y 333.82,Z 609.355,A -85,B 0,C 180,E1 13840.627,E2 13840.627} C_VEL
LIN {X 0,Y 331.462,Z 631.455,A -85,B 0,C 180,E1 13844.769,E2 13844.769} C_VEL
LIN {X 0,Y 329.754,Z 648.446,A -85,B 0,C 180,E1 13849.413,E2 13849.413} C_VEL
LIN {X 0,Y 329.017,Z 659.458,A -85,B 0,C 180,E1 13854.053,E2 13854.053} C_VEL
LIN {X 0,Y 329.039,Z 665.552,A -85,B 0,C 180,E1 13858.678,E2 13858.678} C_VEL
LIN {X 0,Y 329.408,Z 667.194,A -85,B 0,C 180,E1 13862.63,E2 13862.63} C_VEL
LIN {X 0,Y 330.9,Z 664.16,A -85,B 0,C 180,E1 13867.885,E2 13867.885} C_VEL
LIN {X 0,Y 333.054,Z 656.156,A -85,B 0,C 180,E1 13872.567,E2 13872.567} C_VEL
LIN {X 0,Y 336.282,Z 642.785,A -85,B 0,C 180,E1 13877.012,E2 13877.012} C_VEL
LIN {X 0,Y 340.097,Z 623.264,A -85,B 0,C 180,E1 13881.2,E2 13881.2} C_VEL
LIN {X 0,Y 343.869,Z 599.428,A -85,B 0,C 180,E1 13884.623,E2 13884.623} C_VEL
LIN {X 0,Y 347.187,Z 570.114,A -85,B 0,C 180,E1 13887.422,E2 13887.422} C_VEL
LIN {X 0,Y 349.279,Z 538.229,A -85,B 0,C 180,E1 13889.331,E2 13889.331} C_VEL
LIN {X 0,Y 348.481,Z 527.83,A -85,B 0,C 180,E1 13889.951,E2 13889.951} C_VEL
LIN {X 0,Y 345.033,Z 514.913,A -85,B 0,C 180,E1 13891.301,E2 13891.301} C_VEL
LIN {X 0,Y 347.705,Z 513.59,A -85,B 0,C 180,E1 13891.96,E2 13891.96} C_VEL
LIN {X 0,Y 359.705,Z 535.658,A -85,B 0,C 180,E1 13897.02,E2 13897.02} C_VEL
LIN {X 0,Y 370.599,Z 560.601,A -85,B 0,C 180,E1 13901.355,E2 13901.355} C_VEL
LIN {X 0,Y 374.136,Z 572.7,A -85,B 0,C 180,E1 13903.031,E2 13903.031} C_VEL
LIN {X 0,Y 364.181,Z 617.203,A -85,B 0,C 180,E1 13906.145,E2 13906.145} C_VEL
LIN {X 0,Y 355.151,Z 652.742,A -85,B 0,C 180,E1 13909.647,E2 13909.647} C_VEL
LIN {X 0,Y 345.684,Z 685.834,A -85,B 0,C 180,E1 13914.23,E2 13914.23} C_VEL
LIN {X 0,Y 337.514,Z 714.169,A -85,B 0,C 180,E1 13919.689,E2 13919.689} C_VEL
LIN {X 0,Y 331.522,Z 736.846,A -85,B 0,C 180,E1 13925.729,E2 13925.729} C_VEL
LIN {X 0,Y 327.736,Z 754.846,A -85,B 0,C 180,E1 13932.524,E2 13932.524} C_VEL
LIN {X 0,Y 326.232,Z 766.477,A -85,B 0,C 180,E1 13939.301,E2 13939.301} C_VEL
LIN {X 0,Y 325.909,Z 771.666,A -85,B 0,C 180,E1 13944.668,E2 13944.668} C_VEL
LIN {X 0,Y 326.05,Z 773.437,A -85,B 0,C 180,E1 13950,E2 13950} C_VEL
LIN {X 0,Y 325.912,Z 771.743,A -85,B 0,C 180,E1 13955.331,E2 13955.331} C_VEL
LIN {X 0,Y 326.504,Z 764.834,A -85,B 0,C 180,E1 13961.998,E2 13961.998} C_VEL
LIN {X 0,Y 328.281,Z 751.779,A -85,B 0,C 180,E1 13968.835,E2 13968.835} C_VEL
LIN {X 0,Y 330.553,Z 740.685,A -85,B 0,C 180,E1 13972.955,E2 13972.955} C_VEL
LIN {X 0,Y 328.588,Z 732.592,A -85,B 0,C 180,E1 13975.635,E2 13975.635} C_VEL
LIN {X 0,Y 327.129,Z 723.648,A -85,B 0,C 180,E1 13978.276,E2 13978.276} C_VEL
LIN {X 0,Y 334.082,Z 699.023,A -85,B 0,C 180,E1 13983.723,E2 13983.723} C_VEL
LIN {X 0,Y 342.811,Z 667.67,A -85,B 0,C 180,E1 13988.747,E2 13988.747} C_VEL
LIN {X 0,Y 351.746,Z 633.176,A -85,B 0,C 180,E1 13992.694,E2 13992.694} C_VEL
LIN {X 0,Y 361.361,Z 591.3,A -85,B 0,C 180,E1 13996.086,E2 13996.086} C_VEL
LIN {X 0,Y 364.451,Z 574.943,A -85,B 0,C 180,E1 13997.156,E2 13997.156} C_VEL
LIN {X 0,Y 356.049,Z 552.514,A -85,B 0,C 180,E1 14000.148,E2 14000.148} C_VEL
LIN {X 0,Y 338.203,Z 515.601,A -85,B 0,C 180,E1 14005.881,E2 14005.881} C_VEL
LIN {X 0,Y 322.315,Z 487.943,A -85,B 0,C 180,E1 14011.223,E2 14011.223} C_VEL
LIN {X 0,Y 316.098,Z 477.227,A -85,B 0,C 180,E1 14013.549,E2 14013.549} C_VEL
LIN {X 0,Y 316,Z 476.03,A -85,B 0,C 180,E1 14013.848,E2 14013.848} C_VEL
LIN {X 0,Y 316.354,Z 476.03,A -85,B 0,C 180,E1 14020.432,E2 14020.432} C_VEL
LIN {X 0,Y 316.846,Z 476.03,A -85,B 0,C 180,E1 14028.985,E2 14028.985} C_VEL
LIN {X 0,Y 317.529,Z 476.03,A -85,B 0,C 180,E1 14037.271,E2 14037.271} C_VEL
LIN {X 0,Y 317.536,Z 476.03,A -85,B 0,C 180,E1 14042.737,E2 14042.737} C_VEL
LIN {X 0,Y 316.825,Z 476.03,A -85,B 0,C 180,E1 14051.024,E2 14051.024} C_VEL
LIN {X 0,Y 316.38,Z 476.03,A -85,B 0,C 180,E1 14059.576,E2 14059.576} C_VEL
LIN {X 0,Y 316.078,Z 476.03,A -85,B 0,C 180,E1 14065.542,E2 14065.542} C_VEL
LIN {X 0,Y 315.792,Z 476.03,A -85,B 0,C 180,E1 14071.833,E2 14071.833} C_VEL
LIN {X 0,Y 315.544,Z 476.03,A -85,B 0,C 180,E1 14079.848,E2 14079.848} C_VEL
LIN {X 0,Y 315.497,Z 476.03,A -85,B 0,C 180,E1 14086.684,E2 14086.684} C_VEL
LIN {X 0,Y 317.858,Z 481.625,A -85,B 0,C 180,E1 14087.686,E2 14087.686} C_VEL
LIN {X 0,Y 331.007,Z 502.665,A -85,B 0,C 180,E1 14091.897,E2 14091.897} C_VEL
LIN {X 0,Y 344.778,Z 529.596,A -85,B 0,C 180,E1 14096.235,E2 14096.235} C_VEL
LIN {X 0,Y 355.241,Z 558.575,A -85,B 0,C 180,E1 14100.538,E2 14100.538} C_VEL
LIN {X 0,Y 359.281,Z 576.424,A -85,B 0,C 180,E1 14103.11,E2 14103.11} C_VEL
LIN {X 0,Y 350.715,Z 610.092,A -85,B 0,C 180,E1 14106.632,E2 14106.632} C_VEL
LIN {X 0,Y 341.316,Z 641.135,A -85,B 0,C 180,E1 14111.24,E2 14111.24} C_VEL
LIN {X 0,Y 332.809,Z 666.643,A -85,B 0,C 180,E1 14116.517,E2 14116.517} C_VEL
LIN {X 0,Y 325.903,Z 687.814,A -85,B 0,C 180,E1 14122.66,E2 14122.66} C_VEL
LIN {X 0,Y 321.318,Z 703.706,A -85,B 0,C 180,E1 14129.325,E2 14129.325} C_VEL
LIN {X 0,Y 319.218,Z 713.242,A -85,B 0,C 180,E1 14135.444,E2 14135.444} C_VEL
LIN {X 0,Y 318.067,Z 718.375,A -85,B 0,C 180,E1 14140.977,E2 14140.977} C_VEL
LIN {X 0,Y 317.485,Z 720.446,A -85,B 0,C 180,E1 14147.48,E2 14147.48} C_VEL
LIN {X 0,Y 317.866,Z 719.108,A -85,B 0,C 180,E1 14152.401,E2 14152.401} C_VEL
LIN {X 0,Y 319.412,Z 713.327,A -85,B 0,C 180,E1 14159.143,E2 14159.143} C_VEL
LIN {X 0,Y 322.259,Z 702.945,A -85,B 0,C 180,E1 14165.785,E2 14165.785} C_VEL
LIN {X 0,Y 327.405,Z 687.501,A -85,B 0,C 180,E1 14172.273,E2 14172.273} C_VEL
LIN {X 0,Y 334.996,Z 667.032,A -85,B 0,C 180,E1 14178.285,E2 14178.285} C_VEL
LIN {X 0,Y 344.849,Z 640.472,A -85,B 0,C 180,E1 14183.822,E2 14183.822} C_VEL
LIN {X 0,Y 354.84,Z 610.585,A -85,B 0,C 180,E1 14188.238,E2 14188.238} C_VEL
LIN {X 0,Y 363.806,Z 577.013,A -85,B 0,C 180,E1 14191.835,E2 14191.835} C_VEL
LIN {X 0,Y 363.658,Z 575.956,A -85,B 0,C 180,E1 14192.006,E2 14192.006} C_VEL
LIN {X 0,Y 344.28,Z 585.414,A -85,B 0,C 180,E1 14194.606,E2 14194.606} C_VEL
LIN {X 0,Y 331.857,Z 590.728,A -85,B 0,C 180,E1 14196.697,E2 14196.697} C_VEL
LIN {X 0,Y 328.153,Z 591.55,A -85,B 0,C 180,E1 14197.731,E2 14197.731} C_VEL
LIN {X 0,Y 325.299,Z 618.046,A -85,B 0,C 180,E1 14201.649,E2 14201.649} C_VEL
LIN {X 0,Y 323.044,Z 638.796,A -85,B 0,C 180,E1 14206.098,E2 14206.098} C_VEL
LIN {X 0,Y 321.71,Z 653.305,A -85,B 0,C 180,E1 14210.652,E2 14210.652} C_VEL
LIN {X 0,Y 321.151,Z 663.79,A -85,B 0,C 180,E1 14215.941,E2 14215.941} C_VEL
LIN {X 0,Y 321.454,Z 667.793,A -85,B 0,C 180,E1 14219.996,E2 14219.996} C_VEL
LIN {X 0,Y 322.306,Z 668.036,A -85,B 0,C 180,E1 14225.387,E2 14225.387} C_VEL
LIN {X 0,Y 324.114,Z 663.309,A -85,B 0,C 180,E1 14230.084,E2 14230.084} C_VEL
LIN {X 0,Y 326.907,Z 653.427,A -85,B 0,C 180,E1 14234.753,E2 14234.753} C_VEL
LIN {X 0,Y 330.526,Z 638.466,A -85,B 0,C 180,E1 14239.081,E2 14239.081} C_VEL
LIN {X 0,Y 334.619,Z 618.249,A -85,B 0,C 180,E1 14242.965,E2 14242.965} C_VEL
LIN {X 0,Y 338.558,Z 593.467,A -85,B 0,C 180,E1 14246.192,E2 14246.192} C_VEL
LIN {X 0,Y 341.819,Z 563.893,A -85,B 0,C 180,E1 14248.79,E2 14248.79} C_VEL
LIN {X 0,Y 343.165,Z 532.22,A -85,B 0,C 180,E1 14250.622,E2 14250.622} C_VEL
LIN {X 0,Y 342.015,Z 524.756,A -85,B 0,C 180,E1 14251.407,E2 14251.407} C_VEL
LIN {X 0,Y 345.447,Z 522.281,A -85,B 0,C 180,E1 14252.165,E2 14252.165} C_VEL
LIN {X 0,Y 358.188,Z 547.781,A -85,B 0,C 180,E1 14257.794,E2 14257.794} C_VEL
LIN {X 0,Y 367.885,Z 573.538,A -85,B 0,C 180,E1 14262.077,E2 14262.077} C_VEL
LIN {X 0,Y 366.413,Z 583.315,A -85,B 0,C 180,E1 14262.782,E2 14262.782} C_VEL
LIN {X 0,Y 355.877,Z 627.216,A -85,B 0,C 180,E1 14266.153,E2 14266.153} C_VEL
LIN {X 0,Y 346.365,Z 661.346,A -85,B 0,C 180,E1 14269.889,E2 14269.889} C_VEL
LIN {X 0,Y 336.893,Z 692.443,A -85,B 0,C 180,E1 14274.644,E2 14274.644} C_VEL
LIN {X 0,Y 329.007,Z 718.532,A -85,B 0,C 180,E1 14280.137,E2 14280.137} C_VEL
LIN {X 0,Y 323.196,Z 739.577,A -85,B 0,C 180,E1 14286.222,E2 14286.222} C_VEL
LIN {X 0,Y 319.739,Z 755.726,A -85,B 0,C 180,E1 14292.816,E2 14292.816} C_VEL
LIN {X 0,Y 318.387,Z 765.847,A -85,B 0,C 180,E1 14299.034,E2 14299.034} C_VEL
LIN {X 0,Y 318.044,Z 771.03,A -85,B 0,C 180,E1 14304.536,E2 14304.536} C_VEL
LIN {X 0,Y 318.197,Z 772.784,A -85,B 0,C 180,E1 14310,E2 14310} C_VEL
LIN {X 0,Y 318.047,Z 771.071,A -85,B 0,C 180,E1 14315.463,E2 14315.463} C_VEL
LIN {X 0,Y 318.635,Z 764.274,A -85,B 0,C 180,E1 14322.173,E2 14322.173} C_VEL
LIN {X 0,Y 320.508,Z 751.334,A -85,B 0,C 180,E1 14329.147,E2 14329.147} C_VEL
LIN {X 0,Y 324.564,Z 733.392,A -85,B 0,C 180,E1 14335.564,E2 14335.564} C_VEL
LIN {X 0,Y 327.129,Z 723.648,A -85,B 0,C 180,E1 14338.276,E2 14338.276} C_VEL
LIN {X 0,Y 326.184,Z 714.182,A -85,B 0,C 180,E1 14340.861,E2 14340.861} C_VEL
LIN {X 0,Y 325.491,Z 703.783,A -85,B 0,C 180,E1 14343.347,E2 14343.347} C_VEL
LIN {X 0,Y 334.127,Z 674.506,A -85,B 0,C 180,E1 14348.447,E2 14348.447} C_VEL
LIN {X 0,Y 343.458,Z 640.571,A -85,B 0,C 180,E1 14352.694,E2 14352.694} C_VEL
LIN {X 0,Y 353.233,Z 600.457,A -85,B 0,C 180,E1 14356.219,E2 14356.219} C_VEL
LIN {X 0,Y 357.92,Z 576.946,A -85,B 0,C 180,E1 14357.845,E2 14357.845} C_VEL
LIN {X 0,Y 345.198,Z 545.413,A -85,B 0,C 180,E1 14362.399,E2 14362.399} C_VEL
LIN {X 0,Y 328.747,Z 512.082,A -85,B 0,C 180,E1 14368.025,E2 14368.025} C_VEL
LIN {X 0,Y 314.311,Z 487.672,A -85,B 0,C 180,E1 14373.256,E2 14373.256} C_VEL
LIN {X 0,Y 310.096,Z 481.202,A -85,B 0,C 180,E1 14374.896,E2 14374.896} C_VEL
LIN {X 0,Y 308.147,Z 476.03,A -85,B 0,C 180,E1 14375.865,E2 14375.865} C_VEL
LIN {X 0,Y 308.567,Z 476.03,A -85,B 0,C 180,E1 14382.883,E2 14382.883} C_VEL
LIN {X 0,Y 309.062,Z 476.03,A -85,B 0,C 180,E1 14391.553,E2 14391.553} C_VEL
